(* CODESYS project RobotLibrary.library
   Company: Thorsten Brach
   Description: SRCI Robot Library
   Version: 0.0.0.36
   Placeholder: RobotLibrary
   Author: Thorsten Brach
   Title: RobotLibrary

Project tree, tasks and I/O mapping:
  libraries: RobotLibrarySysDep, 0.0.0.1 (Thorsten Brach); Tc2_Standard, 3.4.5.0 (Beckhoff Automation GmbH)
  Library/
    Constants/
      global variables RobotLibraryConstants
      global variables RobotLibraryDefines
      global variables RobotLibraryEvents
    Enumerations/
      ArmConfig/
        data type ArmConfigElbow
        data type ArmConfigShoulder
        data type ArmConfigWrist
      Events/
        data type RobotLibraryErrorIdEnum
        data type RobotLibraryInfoIdEnum
        data type RobotLibraryWarningIdEnum
      Flag/
        data type SequenceFlag
      Level/
        data type LogLevel
        data type LogLevelEnum
        data type MessageLevel
        data type PriorityLevel
      Miscellaneous/
        data type CircPlane
        data type ControlHalfByte
        data type ErrorReaction
        data type LoadMeasurementSteps
        data type PathChoice
        data type ReferenceElement
        data type Severity
        data type SyncDirection
        data type SyncReaction
        data type TriggerCondition
      Mode/
        data type AbortingMode
        data type BlendingMode
        data type CircMode
        data type CollisionReactionMode
        data type ConnectionMode
        data type DefinitionMode
        data type DetectionMode
        data type ErrorTriggerMode
        data type ExecutionMode
        data type FrameCalculationMode
        data type FunctionMode
        data type InterpolationMode
        data type JogMode
        data type LimitMode
        data type LoadMeasurementMode
        data type LogonMode
        data type MeasuringIoMode
        data type MeasuringUnitMode
        data type OperationMode
        data type OrientationMode
        data type OriMode
        data type ProcessingMode
        data type ResistanceForceMode
        data type ReturnMode
        data type SensorConnectionMode
        data type SingularityAvoidanceMode
        data type SplineMode
        data type StepMode
        data type StopMode
        data type SyncInMode
        data type SyncMode
        data type ThresholdMode
        data type ToolCalculationMode
        data type TrajectoryMode
        data type TransformMode
        data type TriggerModeIo
        data type TriggerModeLimit
        data type TriggerModeMeasurement
        data type TriggerReactionMode
        data type TurnMode
        data type WorkAreaReactionMode
      State/
        data type ActiveCommandRegisterState
        data type BufferStateCmd
        data type BufferStateRsp
        data type CmdMessageState
        data type FsmState
        data type InitializationState
        data type RaPowerState
        data type RaSequenceState
        data type RiState
        data type TelegramState
      Type/
        data type AreaType
        data type AxesGroupParameterCmdEntries
        data type CmdType
        data type ConveyorType
        data type MessageType
        data type ReferenceType
        data type UnitType
    Functions/
      Common/
        function CheckTimeout [ST]
        function SetTimeout [ST]
      Convert/
        DT/
          function DATE_TO_IEC_DATE [ST]
          function IEC_DATE_TO_DATE [ST]
          function IEC_TIME_TO_TIME [ST]
          function IEC_TIMESTAMP_TO_DT [ST]
          function TIME_TO_IEC_TIME [ST]
        Misc/
          function ArmConfigParameterToBytes [ST]
          function BytesToRCSupportedFunctions [ST]
          function ByteToFragmentAction [ST]
          function ByteToVersion [ST]
          function CombineBytesToUint [ST]
          function CombineHalfBytes [ST]
          function CombineHalfSints [ST]
          function DwordToRaStatusWord [ST]
          function FragmentActionToByte [ST]
          function PERCENT_INT_TO_REAL [ST]
          function PlcOptionalCyclicToUint [ST]
          function REAL_TO_PERCENT_INT [ST]
          function REAL_TO_PERCENT_UINT [ST]
          function RobOptionalCyclicToUint [ST]
          function VersionToByte [ST]
          function WordToArmConfigElbow [ST]
          function WordToArmConfigShoulder [ST]
          function WordToArmConfigWrist [ST]
        TO_STRING/
          function AREA_TYPE_TO_STRING [ST]
          function ARM_CONFIG_ELBOW_TO_STRING [ST]
          function ARM_CONFIG_SHOULDER_TO_STRING [ST]
          function ARM_CONFIG_TO_STRING [ST]
          function ARM_CONFIG_WRIST_TO_STRING [ST]
          function BLENDING_MODE_TO_STRING [ST]
          function BYTE_TO_STRING_BIN [ST]
          function CIRC_MODE_TO_STRING [ST]
          function CIRC_PLANE_TO_STRING [ST]
          function CMD_MESSAGE_STATE_TO_STRING [ST]
          function CMD_TYPE_TO_STRING [ST]
          function COLLISION_REACTION_MODE_TO_STRING [ST]
          function CONNECTION_MODE_TO_STRING [ST]
          function CONVEYOR_TYPE_TO_STRING [ST]
          function DATA_ENABLE_SYNC_TO_STRING [ST]
          function DATA_IN_SYNC_TO_STRING [ST]
          function DEFINITION_MODE_TO_STRING [ST]
          function DETECTION_MODE_TO_STRING [ST]
          function ERROR_REACTION_TO_STRING [ST]
          function ERROR_TRIGGER_MODE_TO_STRING [ST]
          function EXECUTION_MODE_TO_STRING [ST]
          function FRAGMENT_ACTION_TO_STRING [ST]
          function FRAME_CALCULATION_MODE_TO_STRING [ST]
          function IEC_DATE_TO_STRING [ST]
          function IEC_TIME_TO_STRING [ST]
          function INTERPOLATION_MODE_TO_STRING [ST]
          function JOG_MODE_TO_STRING [ST]
          function LIMIT_MODE_TO_STRING [ST]
          function LOAD_MEASUREMENT_MODE_TO_STRING [ST]
          function LOAD_MEASUREMENT_STEPS_TO_STRING [ST]
          function LOG_LEVEL_TO_STRING [ST]
          function LOGON_MODE_TO_STRING [ST]
          function MEASUREING_UNIT_MODE_TO_STRING [ST]
          function MESSAGE_TYPE_TO_STRING [ST]
          function ORI_MODE_TO_STRING [ST]
          function REFERENCE_TYPE_TO_STRING [ST]
          function SENSOR_CONNECTION_MODE_TO_STRING [ST]
          function SEVERITY_TO_STRING [ST]
          function SINGULARITY_AVOIDANCE_MODE_TO_STRING [ST]
          function SPLINE_MODE_TO_STRING [ST]
          function STEP_MODE_TO_STRING [ST]
          function STOP_MODE_TO_STRING [ST]
          function SYNC_IN_MODE_TO_STRING [ST]
          function SYNC_REACTION_TO_STRING [ST]
          function TELEGRAM_CONTROL_TO_STRING [ST]
          function TELEGRAM_STATE_TO_STRING [ST]
          function THRESHOLD_MODE_TO_STRING [ST]
          function TOOL_CALCULATION_MODE_TO_STRING [ST]
          function TRANSFORM_MODE_TO_STRING [ST]
          function TRIGGER_CONDITION_TO_STRING [ST]
          function TRIGGER_MODE_IO_TO_STRING [ST]
          function TRIGGER_MODE_MEASUREMENT_TO_STRING [ST]
          function TRIGGER_REACTION_MODE_TO_STRING [ST]
          function TURN_MODE_TO_STRING [ST]
          function WORD_TO_STRING_BIN [ST]
          function WORD_TO_STRING_HEX [ST]
          function WORK_AREA_REACTION_MODE_TO_STRING [ST]
      String/
        function StrPadRight [ST]
        function StrReplace [ST]
      Swap/
        function GetHalfeByteHi [ST]
        function GetHalfeByteLo [ST]
        function SwapBytes [ST]
        function SwapDword [ST]
        function SwapIecDate [ST]
        function SwapIecTime [ST]
        function SwapInt [ST]
        function SwapReal [ST]
        function SwapUdint [ST]
        function SwapUint [ST]
        function SwapWord [ST]
    Interfaces/
      interface IMessageLogger: AddMessageLog, AddSystemLog
      interface IRobotLibraryCommandFB: CallBack, CommandData
    Parameter/
      global variables RobotLibraryParameter
    POUs/
      _internal/
        function block ActiveCommandRegisterFB [ST]: AddCmd, AddRsp, CreateUniqueID, FB_init, ManageRegister, NotifyParameterChanged, OnOnlineChange, RemoveCmd, UpdateExecutionOrderList
        function block AxesGroupMessageLogFB [ST]: AddMessage, AddSystemLog, DeleteMessages, DeleteSystemLogs
        function block RobotLibraryBaseEnableFB [ST]: FSM, OnCall, OnExecCancel, OnExecErrorClear, OnExecRun, OnExecStart, Reset
        function block RobotLibraryBaseExecuteFB [ST]: FSM, OnCall, OnExecCancel, OnExecErrorClear, OnExecRun, OnExecStart, Reset
        function block RobotLibraryBaseFB [ST]: CallBack, CheckFunctionSupported, CheckParameterChanged, CheckParameterValid, CreateCommandPayload, OnCall, OnOnlineChange, ParseResponsePayload, Reset
        function block RobotLibraryLogFB [ST]: CreateLogMessage, CreateLogMessagePara1, CreateLogMessagePara2, CreateLogMessagePara3, CreateLogMessagePara4, CreateLogMessagePara5, CreateLogMessagePara6, MyType
        function block RobotLibraryRecvDataFB [ST]: GetArmConfig, GetBool, GetByte, GetDataBlock, GetDataInSync, GetDword, GetFragmentAction, GetHalfeByte1, GetHalfeByte2, GetIecDate, GetIecTime, GetInt, GetReal, GetSint, GetString, GetTrackingStatus, GetTurnNumbers, GetUdint, GetUint, GetUsint, GetWord, Reset
        function block RobotLibrarySendDataFB [ST]: AddArmConfig, AddBool, AddByte, AddDataBlock, AddDataEnableSync, AddDataInSync, AddDword, AddHalfBytes, AddIecDate, AddIecTime, AddInt, AddReal, AddSint, AddString, AddTime, AddTurnNumber, AddUdint, AddUint, AddUsint, Reset
      Additional/
        MC_AbortMeasuringInput/
          Structures/
            data type AbortMeasuringInputOutCmd
            data type AbortMeasuringInputParCmd
            data type AbortMeasuringInputRecvData
            data type AbortMeasuringInputSendData
          function block MC_AbortMeasuringInputFB [ST]: CheckFunctionSupported, CheckParameterChanged, CreateCommandPayload, CreateCommandPayloadLog, FB_init, OnCall, ParseResponsePayload, ParseResponsePayloadLog, Reset
        MC_ActivateNextCommand/
          Structures/
            data type ActivateNextCommandOutCmd
            data type ActivateNextCommandParCmd
            data type ActivateNextCommandRecvData
            data type ActivateNextCommandSendData
          function block MC_ActivateNextCommandFB [ST]: CheckFunctionSupported, CheckParameterChanged, CreateCommandPayload, CreateCommandPayloadLog, FB_init, OnCall, ParseResponsePayload, ParseResponsePayloadLog, Reset
        MC_AvoidSingularity/
          Structures/
            data type AvoidSingularityOutCmd
            data type AvoidSingularityParCmd
            data type AvoidSingularityRecvData
            data type AvoidSingularitySendData
          function block MC_AvoidSingularityFB [ST]: CheckFunctionSupported, CheckParameterChanged, CreateCommandPayload, CreateCommandPayloadLog, FB_init, OnCall, ParseResponsePayload, ParseResponsePayloadLog, Reset
        MC_BrakeTest/
          Structures/
            data type BrakeTestOutCmd
            data type BrakeTestParCmd
            data type BrakeTestRecvData
            data type BrakeTestSendData
          function block MC_BrakeTestFB [ST]: CheckFunctionSupported, CheckParameterChanged, CreateCommandPayload, CreateCommandPayloadLog, FB_init, OnCall, ParseResponsePayload, ParseResponsePayloadLog, Reset
        MC_CallSubprogram/
          Structures/
            data type CallSubprogramOutCmd
            data type CallSubprogramParCmd
            data type CallSubprogramRecvData
            data type CallSubprogramSendData
          function block MC_CallSubprogramFB [ST]: CheckFunctionSupported, CheckParameterChanged, CreateCommandPayload, CreateCommandPayloadLog, FB_init, OnCall, ParseResponsePayload, ParseResponsePayloadLog, Reset
        MC_CollisionDetection/
          Structures/
            data type CollisionDetectionOutCmd
            data type CollisionDetectionParCmd
            data type CollisionDetectionRecvData
            data type CollisionDetectionSendData
          function block MC_CollisionDetectionFB [ST]: CheckFunctionSupported, CheckParameterChanged, CreateCommandPayload, CreateCommandPayloadLog, FB_init, OnCall, ParseResponsePayload, ParseResponsePayloadLog, Reset
        MC_ExchangeConfiguration/
          Structures/
            data type ExchangeConfigurationOutCmd
            data type ExchangeConfigurationParCmd
            data type ExchangeConfigurationRecvData
            data type ExchangeConfigurationSendData
          function block MC_ExchangeConfigurationFB [ST]: CheckFunctionSupported, CheckParameterChanged, CreateCommandPayload, CreateCommandPayloadLog, FB_init, OnCall, ParseResponsePayload, ParseResponsePayloadLog, Reset
        MC_FreeDrive/
          Structures/
            data type FreeDriveOutCmd
            data type FreeDriveParCmd
            data type FreeDriveRecvData
            data type FreeDriveSendData
          function block MC_FreeDriveFB [ST]: CheckFunctionSupported, CheckParameterChanged, CreateCommandPayload, CreateCommandPayloadLog, FB_init, OnCall, ParseResponsePayload, ParseResponsePayloadLog, Reset
        MC_MeasuringInput/
          Structures/
            data type MeasuringInputOutCmd
            data type MeasuringInputParCmd
            data type MeasuringInputRecvData
            data type MeasuringInputSendData
          function block MC_MeasuringInputFB [ST]: CheckFunctionSupported, CheckParameterChanged, CreateCommandPayload, CreateCommandPayloadLog, FB_init, OnCall, ParseResponsePayload, ParseResponsePayloadLog, Reset
        MC_OpenBrake/
          Structures/
            data type OpenBrakeOutCmd
            data type OpenBrakeParCmd
            data type OpenBrakeRecvData
            data type OpenBrakeSendData
          function block MC_OpenBrakeFB [ST]: CheckFunctionSupported, CheckParameterChanged, CreateCommandPayload, CreateCommandPayloadLog, FB_init, OnCall, ParseResponsePayload, ParseResponsePayloadLog, Reset
        MC_PathAccuracyMode/
          Structures/
            data type PathAccuracyModeOutCmd
            data type PathAccuracyModeParCmd
            data type PathAccuracyModeRecvData
            data type PathAccuracyModeSendData
          function block MC_PathAccuracyModeFB [ST]: CheckFunctionSupported, CheckParameterChanged, CreateCommandPayload, CreateCommandPayloadLog, FB_init, OnCall, ParseResponsePayload, ParseResponsePayloadLog, Reset
        MC_ReadCallSubprogramCyclic/
          Structures/
            data type ReadCallSubprogramCyclicOutCmd
            data type ReadCallSubprogramCyclicParCmd
          function block MC_ReadCallSubprogramCyclicFB [ST]: CheckFunctionSupported, FB_init, OnCall
        MC_ShiftPosition/
          Structures/
            data type ShiftPositionOutCmd
            data type ShiftPositionParCmd
            data type ShiftPositionRecvData
            data type ShiftPositionSendData
          function block MC_ShiftPositionFB [ST]: CheckFunctionSupported, CheckParameterChanged, CreateCommandPayload, CreateCommandPayloadLog, FB_init, OnCall, ParseResponsePayload, ParseResponsePayloadLog, Reset
        MC_SoftSwitchTcp/
          Structures/
            data type SoftSwitchTcpOutCmd
            data type SoftSwitchTcpParCmd
            data type SoftSwitchTcpRecvData
            data type SoftSwitchTcpSendData
          function block MC_SoftSwitchTcpFB [ST]: CheckFunctionSupported, CheckParameterChanged, CreateCommandPayload, CreateCommandPayloadLog, FB_init, OnCall, ParseResponsePayload, ParseResponsePayloadLog, Reset
        MC_StopSubprogram/
          Structures/
            data type StopSubprogramOutCmd
            data type StopSubprogramParCmd
            data type StopSubprogramRecvData
            data type StopSubprogramSendData
          function block MC_StopSubprogramFB [ST]: CheckFunctionSupported, CheckParameterChanged, CreateCommandPayload, CreateCommandPayloadLog, FB_init, OnCall, ParseResponsePayload, ParseResponsePayloadLog, Reset
        MC_UnitMeasurement/
          Structures/
            data type UnitMeasurementOutCmd
            data type UnitMeasurementParCmd
            data type UnitMeasurementRecvData
            data type UnitMeasurementSendData
          function block MC_UnitMeasurementFB [ST]: CheckFunctionSupported, CheckParameterChanged, CreateCommandPayload, CreateCommandPayloadLog, FB_init, OnCall, ParseResponsePayload, ParseResponsePayloadLog, Reset
        MC_WriteCallSubprogramCyclic/
          Structures/
            data type WriteCallSubprogramCyclicOutCmd
            data type WriteCallSubprogramCyclicParCmd
          function block MC_WriteCallSubprogramCyclicFB [ST]: CheckFunctionSupported, FB_init, OnCall
      AdvancedMove/
        MC_MoveApproachDirect/
          Structures/
            data type MoveApproachDirectOutCmd
            data type MoveApproachDirectParCmd
            data type MoveApproachDirectRecvData
            data type MoveApproachDirectSendData
          function block MC_MoveApproachDirectFB [ST]: CheckFunctionSupported, CheckParameterChanged, CreateCommandPayload, CreateCommandPayloadLog, FB_init, OnCall, ParseResponsePayload, ParseResponsePayloadLog, Reset
        MC_MoveApproachLinear/
          Structures/
            data type MoveApproachLinearOutCmd
            data type MoveApproachLinearParCmd
            data type MoveApproachLinearRecvData
            data type MoveApproachLinearSendData
          function block MC_MoveApproachLinearFB [ST]: CheckFunctionSupported, CheckParameterChanged, CreateCommandPayload, CreateCommandPayloadLog, FB_init, OnCall, ParseResponsePayload, ParseResponsePayloadLog, Reset
        MC_MoveAxesRelative/
          Structures/
            data type MoveAxesRelativeOutCmd
            data type MoveAxesRelativeParCmd
            data type MoveAxesRelativeRecvData
            data type MoveAxesRelativeSendData
          function block MC_MoveAxesRelativeFB [ST]: CheckFunctionSupported, CheckParameterChanged, CreateCommandPayload, CreateCommandPayloadLog, FB_init, OnCall, ParseResponsePayload, ParseResponsePayloadLog, Reset
        MC_MoveCircularAbsolute/
          Structures/
            data type MoveCircularAbsoluteOutCmd
            data type MoveCircularAbsoluteParCmd
            data type MoveCircularAbsoluteRecvData
            data type MoveCircularAbsoluteSendData
          function block MC_MoveCircularAbsoluteFB [ST]: CheckFunctionSupported, CheckParameterChanged, CreateCommandPayload, CreateCommandPayloadLog, FB_init, OnCall, ParseResponsePayload, ParseResponsePayloadLog, Reset
        MC_MoveCircularCamFB/
          Structures/
            data type MoveCircularCamOutCmd
            data type MoveCircularCamParCmd
            data type MoveCircularCamRecvData
            data type MoveCircularCamSendData
          function block MC_MoveCircularCamFB [ST]: CheckFunctionSupported, CheckParameterChanged, CreateCommandPayload, CreateCommandPayloadLog, FB_init, OnCall, ParseResponsePayload, ParseResponsePayloadLog, Reset
        MC_MoveCircularRelative/
          Structures/
            data type MoveCircularRelativeOutCmd
            data type MoveCircularRelativeParCmd
            data type MoveCircularRelativeRecvData
            data type MoveCircularRelativeSendData
          function block MC_MoveCircularRelativeFB [ST]: CheckFunctionSupported, CheckParameterChanged, CreateCommandPayload, CreateCommandPayloadLog, FB_init, OnCall, ParseResponsePayload, ParseResponsePayloadLog, Reset
        MC_MoveDepartDirect/
          Structures/
            data type MoveDepartDirectOutCmd
            data type MoveDepartDirectParCmd
            data type MoveDepartDirectRecvData
            data type MoveDepartDirectSendData
          function block MC_MoveDepartDirectFB [ST]: CheckFunctionSupported, CheckParameterChanged, CreateCommandPayload, CreateCommandPayloadLog, FB_init, OnCall, ParseResponsePayload, ParseResponsePayloadLog, Reset
        MC_MoveDepartLinear/
          Structures/
            data type MoveDepartLinearOutCmd
            data type MoveDepartLinearParCmd
            data type MoveDepartLinearRecvData
            data type MoveDepartLinearSendData
          function block MC_MoveDepartLinearFB [ST]: CheckFunctionSupported, CheckParameterChanged, CreateCommandPayload, CreateCommandPayloadLog, FB_init, OnCall, ParseResponsePayload, ParseResponsePayloadLog, Reset
        MC_MoveDirectOffset/
          Structures/
            data type MoveDirectOffsetOutCmd
            data type MoveDirectOffsetParCmd
            data type MoveDirectOffsetRecvData
            data type MoveDirectOffsetSendData
          function block MC_MoveDirectOffsetFB [ST]: CheckFunctionSupported, CheckParameterChanged, CreateCommandPayload, CreateCommandPayloadLog, FB_init, OnCall, ParseResponsePayload, ParseResponsePayloadLog, Reset
        MC_MoveDirectRelative/
          Structures/
            data type MoveDirectRelativeOutCmd
            data type MoveDirectRelativeParCmd
            data type MoveDirectRelativeRecvData
            data type MoveDirectRelativeSendData
          function block MC_MoveDirectRelativeFB [ST]: CheckFunctionSupported, CheckParameterChanged, CreateCommandPayload, CreateCommandPayloadLog, FB_init, OnCall, ParseResponsePayload, ParseResponsePayloadLog, Reset
        MC_MoveLinearAbsoluteJ/
          Structures/
            data type MoveLinearAbsoluteJOutCmd
            data type MoveLinearAbsoluteJParCmd
            data type MoveLinearAbsoluteJRecvData
            data type MoveLinearAbsoluteJSendData
          function block MC_MoveLinearAbsoluteJFB [ST]: CheckFunctionSupported, CheckParameterChanged, CreateCommandPayload, CreateCommandPayloadLog, FB_init, OnCall, ParseResponsePayload, ParseResponsePayloadLog, Reset
        MC_MoveLinearCam/
          Structures/
            data type MoveLinearCamOutCmd
            data type MoveLinearCamParCmd
            data type MoveLinearCamRecvData
            data type MoveLinearCamSendData
          function block MC_MoveLinearCamFB [ST]: CheckFunctionSupported, CheckParameterChanged, CreateCommandPayload, CreateCommandPayloadLog, FB_init, OnCall, ParseResponsePayload, ParseResponsePayloadLog, Reset
        MC_MoveLinearOffset/
          Structures/
            data type MoveLinearOffsetOutCmd
            data type MoveLinearOffsetParCmd
            data type MoveLinearOffsetRecvData
            data type MoveLinearOffsetSendData
          function block MC_MoveLinearOffsetFB [ST]: CheckFunctionSupported, CheckParameterChanged, CreateCommandPayload, CreateCommandPayloadLog, FB_init, OnCall, ParseResponsePayload, ParseResponsePayloadLog, Reset
        MC_MoveLinearRelative/
          Structures/
            data type MoveLinearRelativeOutCmd
            data type MoveLinearRelativeParCmd
            data type MoveLinearRelativeRecvData
            data type MoveLinearRelativeSendData
          function block MC_MoveLinearRelativeFB [ST]: CheckFunctionSupported, CheckParameterChanged, CreateCommandPayload, CreateCommandPayloadLog, FB_init, OnCall, ParseResponsePayload, ParseResponsePayloadLog, Reset
        MC_MovePickPlaceDirect/
          Structures/
            data type MovePickPlaceDirectOutCmd
            data type MovePickPlaceDirectParCmd
            data type MovePickPlaceDirectRecvData
            data type MovePickPlaceDirectSendData
          function block MC_MovePickPlaceDirectFB [ST]: CheckFunctionSupported, CheckParameterChanged, CreateCommandPayload, CreateCommandPayloadLog, FB_init, OnCall, ParseResponsePayload, ParseResponsePayloadLog, Reset
        MC_MovePickPlaceLinear/
          Structures/
            data type MovePickPlaceLinearOutCmd
            data type MovePickPlaceLinearParCmd
            data type MovePickPlaceLinearRecvData
            data type MovePickPlaceLinearSendData
          function block MC_MovePickPlaceLinearFB [ST]: CheckFunctionSupported, CheckParameterChanged, CreateCommandPayload, CreateCommandPayloadLog, FB_init, OnCall, ParseResponsePayload, ParseResponsePayloadLog, Reset
      BasicMove/
        MC_ChangeSpeedOverride/
          Structures/
            data type ChangeSpeedOverrideOutCmd
            data type ChangeSpeedOverrideParCmd
            data type ChangeSpeedOverrideRecvData
            data type ChangeSpeedOverrideSendData
          function block MC_ChangeSpeedOverrideFB [ST]: CheckFunctionSupported, CheckParameterChanged, CreateCommandPayload, CreateCommandPayloadLog, FB_init, OnCall, ParseResponsePayload, ParseResponsePayloadLog, Reset
        MC_GroupContinue/
          Structures/
            data type GroupContinueOutCmd
            data type GroupContinueParCmd
            data type GroupContinueRecvData
            data type GroupContinueSendData
          function block MC_GroupContinueFB [ST]: CheckFunctionSupported, CheckParameterChanged, CreateCommandPayload, CreateCommandPayloadLog, FB_init, OnCall, ParseResponsePayload, ParseResponsePayloadLog, Reset
        MC_GroupInterrupt/
          Structures/
            data type GroupInterruptOutCmd
            data type GroupInterruptParCmd
            data type GroupInterruptRecvData
            data type GroupInterruptSendData
          function block MC_GroupInterruptFB [ST]: CheckFunctionSupported, CheckParameterChanged, CreateCommandPayload, CreateCommandPayloadLog, FB_init, OnCall, ParseResponsePayload, ParseResponsePayloadLog, Reset
        MC_GroupJog/
          Structures/
            data type GroupJogOutCmd
            data type GroupJogParCmd
            data type GroupJogRecvData
            data type GroupJogSendData
          function block MC_GroupJogFB [ST]: CheckFunctionSupported, CheckParameterChanged, CreateCommandPayload, CreateCommandPayloadLog, FB_init, OnCall, ParseResponsePayload, ParseResponsePayloadLog, Reset
        MC_GroupStop/
          Structures/
            data type GroupStopOutCmd
            data type GroupStopParCmd
            data type GroupStopRecvData
            data type GroupStopSendData
          function block MC_GroupStopFB [ST]: CheckFunctionSupported, CheckParameterChanged, CreateCommandPayload, CreateCommandPayloadLog, FB_init, OnCall, ParseResponsePayload, ParseResponsePayloadLog, Reset
        MC_MoveAxesAbsolute/
          Structures/
            data type MoveAxesAbsoluteOutCmd
            data type MoveAxesAbsoluteParCmd
            data type MoveAxesAbsoluteRecvData
            data type MoveAxesAbsoluteSendData
          function block MC_MoveAxesAbsoluteFB [ST]: CheckFunctionSupported, CheckParameterChanged, CreateCommandPayload, CreateCommandPayloadLog, FB_init, OnCall, ParseResponsePayload, ParseResponsePayloadLog, Reset
        MC_MoveDirectAbsolute/
          Structures/
            data type MoveDirectAbsoluteOutCmd
            data type MoveDirectAbsoluteParCmd
            data type MoveDirectAbsoluteRecvData
            data type MoveDirectAbsoluteSendData
          function block MC_MoveDirectAbsoluteFB [ST]: CheckFunctionSupported, CheckParameterChanged, CreateCommandPayload, CreateCommandPayloadLog, FB_init, OnCall, ParseResponsePayload, ParseResponsePayloadLog, Reset
        MC_MoveLinearAbsolute/
          Structures/
            data type MoveLinearAbsoluteOutCmd
            data type MoveLinearAbsoluteParCmd
            data type MoveLinearAbsoluteRecvData
            data type MoveLinearAbsoluteSendData
          function block MC_MoveLinearAbsoluteFB [ST]: CheckFunctionSupported, CheckParameterChanged, CreateCommandPayload, CreateCommandPayloadLog, FB_init, OnCall, ParseResponsePayload, ParseResponsePayloadLog, Reset
        MC_ReturnToPrimary/
          Structures/
            data type ReturnToPrimaryOutCmd
            data type ReturnToPrimaryParCmd
            data type ReturnToPrimaryRecvData
            data type ReturnToPrimarySendData
          function block MC_ReturnToPrimaryFB [ST]: CheckFunctionSupported, CheckParameterChanged, CreateCommandPayload, CreateCommandPayloadLog, FB_init, OnCall, ParseResponsePayload, ParseResponsePayloadLog, Reset
      Calculation/
        MC_CalculateCartesianPosition/
          Structures/
            data type CalculateCartesianPositionOutCmd
            data type CalculateCartesianPositionParCmd
            data type CalculateCartesianPositionRecvData
            data type CalculateCartesianPositionSendData
          function block MC_CalculateCartesianPositionFB [ST]: CheckFunctionSupported, CheckParameterChanged, CreateCommandPayload, CreateCommandPayloadLog, FB_init, OnCall, ParseResponsePayload, ParseResponsePayloadLog, Reset
        MC_CalculateForwardKinematic/
          Structures/
            data type CalculateForwardKinematicOutCmd
            data type CalculateForwardKinematicParCmd
            data type CalculateForwardKinematicRecvData
            data type CalculateForwardKinematicSendData
          function block MC_CalculateForwardKinematicFB [ST]: CheckFunctionSupported, CheckParameterChanged, CreateCommandPayload, CreateCommandPayloadLog, FB_init, OnCall, ParseResponsePayload, ParseResponsePayloadLog, Reset
        MC_CalculateFrame/
          Structures/
            data type CalculateFrameOutCmd
            data type CalculateFrameParCmd
            data type CalculateFrameRecvData
            data type CalculateFrameSendData
          function block MC_CalculateFrameFB [ST]: CheckFunctionSupported, CheckParameterChanged, CreateCommandPayload, CreateCommandPayloadLog, FB_init, OnCall, ParseResponsePayload, ParseResponsePayloadLog, Reset
        MC_CalculateInverseKinematic/
          Structures/
            data type CalculateInverseKinematicOutCmd
            data type CalculateInverseKinematicParCmd
            data type CalculateInverseKinematicRecvData
            data type CalculateInverseKinematicSendData
          function block MC_CalculateInverseKinematicFB [ST]: CheckFunctionSupported, CheckParameterChanged, CreateCommandPayload, CreateCommandPayloadLog, FB_init, OnCall, ParseResponsePayload, ParseResponsePayloadLog, Reset
        MC_CalculateTool/
          Structures/
            data type CalculateToolOutCmd
            data type CalculateToolParCmd
            data type CalculateToolRecvData
            data type CalculateToolSendData
          function block MC_CalculateToolFB [ST]: CheckFunctionSupported, CheckParameterChanged, CreateCommandPayload, CreateCommandPayloadLog, FB_init, OnCall, ParseResponsePayload, ParseResponsePayloadLog, Reset
        MC_LoadMeasurementAutomatic/
          Structures/
            data type LoadMeasurementAutomaticOutCmd
            data type LoadMeasurementAutomaticParCmd
            data type LoadMeasurementAutomaticRecvData
            data type LoadMeasurementAutomaticSendData
          function block MC_LoadMeasurementAutomaticFB [ST]: CheckFunctionSupported, CheckParameterChanged, CreateCommandPayload, CreateCommandPayloadLog, FB_init, OnCall, ParseResponsePayload, ParseResponsePayloadLog, Reset
        MC_LoadMeasurementSequential/
          Structures/
            data type LoadMeasurementSequentialOutCmd
            data type LoadMeasurementSequentialParCmd
            data type LoadMeasurementSequentialRecvData
            data type LoadMeasurementSequentialSendData
          function block MC_LoadMeasurementSequentialFB [ST]: CheckFunctionSupported, CheckParameterChanged, CreateCommandPayload, CreateCommandPayloadLog, FB_init, OnCall, ParseResponsePayload, ParseResponsePayloadLog, Reset
      ConveyorTracking/
        MC_ActivateConveyorTracking/
          Structures/
            data type ActivateConveyorTrackingOutCmd
            data type ActivateConveyorTrackingParCmd
            data type ActivateConveyorTrackingRecvData
            data type ActivateConveyorTrackingSendData
          function block MC_ActivateConveyorTrackingFB [ST]: CheckFunctionSupported, CheckParameterChanged, CreateCommandPayload, CreateCommandPayloadLog, FB_init, OnCall, ParseResponsePayload, ParseResponsePayloadLog, Reset
        MC_ConfigureConveyor/
          Structures/
            data type ConfigureConveyorOutCmd
            data type ConfigureConveyorParCmd
            data type ConfigureConveyorRecvData
            data type ConfigureConveyorSendData
          function block MC_ConfigureConveyorFB [ST]: CheckFunctionSupported, CheckParameterChanged, CreateCommandPayload, CreateCommandPayloadLog, FB_init, OnCall, ParseResponsePayload, ParseResponsePayloadLog, Reset
        MC_RedefineTrackingPos/
          Structures/
            data type RedefineTrackingPosOutCmd
            data type RedefineTrackingPosParCmd
            data type RedefineTrackingPosRecvData
            data type RedefineTrackingPosSendData
          function block MC_RedefineTrackingPosFB [ST]: CheckFunctionSupported, CheckParameterChanged, CreateCommandPayload, CreateCommandPayloadLog, FB_init, OnCall, ParseResponsePayload, ParseResponsePayloadLog, Reset
        MC_SyncToConveyor/
          Structures/
            data type SyncToConveyorOutCmd
            data type SyncToConveyorParCmd
            data type SyncToConveyorRecvData
            data type SyncToConveyorSendData
          function block MC_SyncToConveyorFB [ST]: CheckFunctionSupported, CheckParameterChanged, CreateCommandPayload, CreateCommandPayloadLog, FB_init, OnCall, ParseResponsePayload, ParseResponsePayloadLog, Reset
      ForceControl/
        MC_ForceControl/
          Structures/
            data type ForceControlOutCmd
            data type ForceControlParCmd
            data type ForceControlRecvData
            data type ForceControlSendData
          function block MC_ForceControlFB [ST]: CheckFunctionSupported, CheckParameterChanged, CreateCommandPayload, CreateCommandPayloadLog, FB_init, OnCall, ParseResponsePayload, ParseResponsePayloadLog, Reset
        MC_ForceLimit/
          Structures/
            data type ForceLimitOutCmd
            data type ForceLimitParCmd
            data type ForceLimitRecvData
            data type ForceLimitSendData
          function block MC_ForceLimitFB [ST]: CheckFunctionSupported, CheckParameterChanged, CreateCommandPayload, CreateCommandPayloadLog, FB_init, OnCall, ParseResponsePayload, ParseResponsePayloadLog, Reset
        MC_ReadActualForce/
          Structures/
            data type ReadActualForceOutCmd
            data type ReadActualForceParCmd
            data type ReadActualForceRecvData
            data type ReadActualForceSendData
          function block MC_ReadActualForceFB [ST]: CheckFunctionSupported, CheckParameterChanged, CreateCommandPayload, CreateCommandPayloadLog, FB_init, OnCall, ParseResponsePayload, ParseResponsePayloadLog, Reset
      General/
        MC_CreateServerLog_ToDo/
          function block MC_CreateServerLog_ToDo [ST]: FB_init
        MC_EnableRobot/
          Structures/
            data type EnableRobotOutCmd
            data type EnableRobotParCmd
            data type EnableRobotRecvData
            data type EnableRobotSendData
          function block MC_EnableRobotFB [ST]: CheckFunctionSupported, CheckParameterChanged, CreateCommandPayload, CreateCommandPayloadLog, FB_init, OnCall, ParseResponsePayload, ParseResponsePayloadLog, Reset
        MC_GroupReset/
          Structures/
            data type GroupResetOutCmd
            data type GroupResetParCmd
            data type GroupResetRecvData
            data type GroupResetSendData
          function block MC_GroupResetFB [ST]: CheckFunctionSupported, CheckParameterChanged, CreateCommandPayload, CreateCommandPayloadLog, FB_init, OnCall, ParseResponsePayload, ParseResponsePayloadLog, Reset
        MC_ReadServerLog_ToDo/
          function block MC_ReadServerLog [ST]: FB_init
        MC_RestartController/
          Structures/
            data type RestartControllerOutCmd
            data type RestartControllerParCmd
            data type RestartControllerRecvData
            data type RestartControllerSendData
          function block MC_RestartControllerFB [ST]: CheckFunctionSupported, CheckParameterChanged, CreateCommandPayload, CreateCommandPayloadLog, FB_init, OnCall, ParseResponsePayload, ParseResponsePayloadLog, Reset
        MC_RobotTask/
          Structures/
            ParCfg/
              Com/
                data type RobotTaskParCfgCom
              Plc/
                data type RobotTaskParCfgPlc
                data type RobotTaskParCfgPlcParameter
              Rob/
                data type RobotTaskParCfgRob
                data type RobotTaskParCfgRobParameter
              data type RobotTaskParCfg
          function block MC_RobotTaskFB [ST]: AxesGroupFromTelegram, AxesGroupFromTelegramCyclic, AxesGroupFromTelegramCyclicOptional, AxesGroupToTelegram, AxesGroupToTelegramCyclic, AxesGroupToTelegramCyclicOptional, AxesGroupToTelegramFooter, AxesGroupToTelegramHeader, AxesGroupToTelegramLogging, AxesGroupToTelegramSequence, CalcTelegramLengthPlcToRob, CreateSendPayload, CreateSendPayloadCyclic, CreateSendPayloadCyclicOptional, CreateSendPayloadFooter, CreateSendPayloadHeader, CreateSendPayloadLogging, CreateSendPayloadSequence, FB_init, HandleAliveBit, HandleAxesGroupAcyclic, HandleAxesGroupCyclic, HandleAxesGroupCyclicOptional, HandleAxesGroupInternalData, HandleAxesGroupMessageLog, HandleAxesGroupParameter, HandleAxesGroupState, HandleInvalidFrames, HandleLifeSign, HandleSeqAck, HandleTelegramStateCtrl, OnCall, OnErrorClear, OnExecRun, ParseRecvPayload, ParseRecvPayloadCyclic, ParseRecvPayloadCyclicOptional, ParseRecvPayloadFooter, ParseRecvPayloadHeader, ParseRecvPayloadLogging, ParseRecvPayloadSequence
        MC_SetOperationMode/
          Structures/
            data type SetOperationModeOutCmd
            data type SetOperationModeParCmd
            data type SetOperationModeRecvData
            data type SetOperationModeSendData
          function block MC_SetOperationModeFB [ST]: CheckFunctionSupported, CheckParameterChanged, CreateCommandPayload, CreateCommandPayloadLog, FB_init, OnCall, ParseResponsePayload, ParseResponsePayloadLog, Reset
        MC_SetSequence/
          Structures/
            data type SetSequenceOutCmd
            data type SetSequenceParCmd
            data type SetSequenceRecvData
            data type SetSequenceSendData
          function block MC_SetSequenceFB [ST]: CheckFunctionSupported, CheckParameterChanged, CreateCommandPayload, CreateCommandPayloadLog, FB_init, OnCall, ParseResponsePayload, ParseResponsePayloadLog, Reset
        MC_SwitchLanguage/
          Structures/
            data type SwitchLanguageOutCmd
            data type SwitchLanguageParCmd
            data type SwitchLanguageRecvData
            data type SwitchLanguageSendData
          function block MC_SwitchLanguageFB [ST]: CheckFunctionSupported, CheckParameterChanged, CreateCommandPayload, CreateCommandPayloadLog, FB_init, OnCall, ParseResponsePayload, ParseResponsePayloadLog, Reset
        MC_UserLogin/
          Structures/
            data type UserLoginOutCmd
            data type UserLoginParCmd
            data type UserLoginRecvData
            data type UserLoginSendData
          function block MC_UserLoginFB [ST]: CheckFunctionSupported, CheckParameterChanged, CreateCommandPayload, CreateCommandPayloadLog, FB_init, OnCall, ParseResponsePayload, ParseResponsePayloadLog, Reset
      Read/
        MC_ReadActualPosition/
          Structures/
            data type ReadActualPositionOutCmd
            data type ReadActualPositionParCmd
            data type ReadActualPositionRecvData
            data type ReadActualPositionSendData
          function block MC_ReadActualPositionFB [ST]: CheckFunctionSupported, CheckParameterChanged, CreateCommandPayload, CreateCommandPayloadLog, FB_init, OnCall, ParseResponsePayload, ParseResponsePayloadLog, Reset
        MC_ReadActualPositionCyclic/
          Structures/
            data type ReadActualPositionCyclicOutCmd
            data type ReadActualPositionCyclicParCmd
          function block MC_ReadActualPositionCyclicFB [ST]: CheckFunctionSupported, CheckParameterChanged, CheckParameterValid, CreateCommandParameterLog, FB_init, OnCall, Reset
        MC_ReadActualTCPVelocity/
          Structures/
            data type ReadActualTCPVelocityOutCmd
            data type ReadActualTCPVelocityParCmd
            data type ReadActualTCPVelocityRecvData
            data type ReadActualTCPVelocitySendData
          function block MC_ReadActualTCPVelocityFB [ST]: CheckFunctionSupported, CheckParameterChanged, CreateCommandPayload, CreateCommandPayloadLog, FB_init, OnCall, ParseResponsePayload, ParseResponsePayloadLog, Reset
        MC_ReadAnalogInput/
          Structures/
            data type ReadAnalogInputOutCmd
            data type ReadAnalogInputParCmd
            data type ReadAnalogInputRecvData
            data type ReadAnalogInputSendData
          function block MC_ReadAnalogInputFB [ST]: CheckFunctionSupported, CheckParameterChanged, CreateCommandPayload, CreateCommandPayloadLog, FB_init, OnCall, ParseResponsePayload, ParseResponsePayloadLog, Reset
        MC_ReadDHParameter/
          Structures/
            data type ReadDHParameterOutCmd
            data type ReadDHParameterParCmd
            data type ReadDHParameterRecvData
            data type ReadDHParameterSendData
          function block MC_ReadDHParameterFB [ST]: CheckFunctionSupported, CheckParameterChanged, CreateCommandPayload, CreateCommandPayloadLog, FB_init, OnCall, ParseResponsePayload, ParseResponsePayloadLog, Reset
        MC_ReadDigitalInputs/
          Structures/
            data type ReadDigitalInputsOutCmd
            data type ReadDigitalInputsParCmd
            data type ReadDigitalInputsRecvData
            data type ReadDigitalInputsSendData
          function block MC_ReadDigitalInputsFB [ST]: CheckFunctionSupported, CheckParameterChanged, CreateCommandPayload, CreateCommandPayloadLog, FB_init, OnCall, ParseResponsePayload, ParseResponsePayloadLog, Reset
        MC_ReadDigitalOutputs/
          Structures/
            data type ReadDigitalOutputsOutCmd
            data type ReadDigitalOutputsParCmd
            data type ReadDigitalOutputsRecvData
            data type ReadDigitalOutputsSendData
          function block MC_ReadDigitalOutputsFB [ST]: CheckFunctionSupported, CheckParameterChanged, CreateCommandPayload, CreateCommandPayloadLog, FB_init, OnCall, ParseResponsePayload, ParseResponsePayloadLog, Reset
        MC_ReadFrameData/
          Structures/
            data type ReadFrameDataOutCmd
            data type ReadFrameDataParCmd
            data type ReadFrameDataRecvData
            data type ReadFrameDataSendData
          function block MC_ReadFrameDataFB [ST]: CheckFunctionSupported, CheckParameterChanged, CreateCommandPayload, CreateCommandPayloadLog, FB_init, OnCall, ParseResponsePayload, ParseResponsePayloadLog, Reset
        MC_ReadIntegers/
          Structures/
            data type ReadIntegersOutCmd
            data type ReadIntegersParCmd
            data type ReadIntegersRecvData
            data type ReadIntegersSendData
          function block MC_ReadIntegersFB [ST]: CheckFunctionSupported, CheckParameterChanged, CreateCommandPayload, CreateCommandPayloadLog, FB_init, OnCall, ParseResponsePayload, ParseResponsePayloadLog, Reset
        MC_ReadLoadData/
          Structures/
            data type ReadLoadDataOutCmd
            data type ReadLoadDataParCmd
            data type ReadLoadDataRecvData
            data type ReadLoadDataSendData
          function block MC_ReadLoadDataFB [ST]: CheckFunctionSupported, CheckParameterChanged, CreateCommandPayload, CreateCommandPayloadLog, FB_init, OnCall, ParseResponsePayload, ParseResponsePayloadLog, Reset
        MC_ReadMessages/
          Structures/
            data type ReadMessagesOutCmd
            data type ReadMessagesParCmd
            data type ReadMessagesRecvData
            data type ReadMessagesSendData
          function block MC_ReadMessagesFB [ST]: CheckFunctionSupported, CheckParameterChanged, CreateCommandPayload, CreateCommandPayloadLog, FB_init, OnCall, ParseResponsePayload, ParseResponsePayloadLog, Reset
        MC_ReadReals/
          Structures/
            data type ReadRealsOutCmd
            data type ReadRealsParCmd
            data type ReadRealsRecvData
            data type ReadRealsSendData
          function block MC_ReadRealsFB [ST]: CheckFunctionSupported, CheckParameterChanged, CreateCommandPayload, CreateCommandPayloadLog, FB_init, OnCall, ParseResponsePayload, ParseResponsePayloadLog, Reset
        MC_ReadRobotData/
          Structures/
            data type ReadRobotDataOutCmd
            data type ReadRobotDataParCmd
            data type ReadRobotDataRecvData
            data type ReadRobotDataSendData
          function block MC_ReadRobotDataFB [ST]: CheckFunctionSupported, CheckParameterChanged, CreateCommandPayload, CreateCommandPayloadLog, FB_init, OnCall, ParseResponsePayload, ParseResponsePayloadLog, Reset
        MC_ReadRobotDefaultDynamics/
          Structures/
            data type ReadRobotDefaultDynamicsOutCmd
            data type ReadRobotDefaultDynamicsParCmd
            data type ReadRobotDefaultDynamicsRecvData
            data type ReadRobotDefaultDynamicsSendData
          function block MC_ReadRobotDefaultDynamicsFB [ST]: CheckFunctionSupported, CheckParameterChanged, CreateCommandPayload, CreateCommandPayloadLog, FB_init, OnCall, ParseResponsePayload, ParseResponsePayloadLog, Reset
        MC_ReadRobotReferenceDynamics/
          Structures/
            data type ReadRobotReferenceDynamicsOutCmd
            data type ReadRobotReferenceDynamicsParCmd
            data type ReadRobotReferenceDynamicsRecvData
            data type ReadRobotReferenceDynamicsSendData
          function block MC_ReadRobotReferenceDynamicsFB [ST]: CheckFunctionSupported, CheckParameterChanged, CreateCommandPayload, CreateCommandPayloadLog, FB_init, OnCall, ParseResponsePayload, ParseResponsePayloadLog, Reset
        MC_ReadRobotSWLimits/
          Structures/
            data type ReadRobotSWLimitsOutCmd
            data type ReadRobotSWLimitsParCmd
            data type ReadRobotSWLimitsRecvData
            data type ReadRobotSWLimitsSendData
          function block MC_ReadRobotSWLimitsFB [ST]: CheckFunctionSupported, CheckParameterChanged, CreateCommandPayload, CreateCommandPayloadLog, FB_init, OnCall, ParseResponsePayload, ParseResponsePayloadLog, Reset
        MC_ReadSystemVariable/
          Structures/
            data type ReadSystemVariableOutCmd
            data type ReadSystemVariableParCmd
            data type ReadSystemVariableRecvData
            data type ReadSystemVariableSendData
          function block MC_ReadSystemVariableFB [ST]: CheckFunctionSupported, CheckParameterChanged, CreateCommandPayload, CreateCommandPayloadLog, FB_init, OnCall, ParseResponsePayload, ParseResponsePayloadLog, Reset
        MC_ReadToolData/
          Structures/
            data type ReadToolDataOutCmd
            data type ReadToolDataParCmd
            data type ReadToolDataRecvData
            data type ReadToolDataSendData
          function block MC_ReadToolDataFB [ST]: CheckFunctionSupported, CheckParameterChanged, CreateCommandPayload, CreateCommandPayloadLog, FB_init, OnCall, ParseResponsePayload, ParseResponsePayloadLog, Reset
      SearchHardstop/
        MC_SearchHardStop/
          Structures/
            data type SearchHardStopOutCmd
            data type SearchHardStopParCmd
            data type SearchHardStopRecvData
            data type SearchHardStopSendData
          function block MC_SearchHardStopFB [ST]: CheckFunctionSupported, CheckParameterChanged, CreateCommandPayload, CreateCommandPayloadLog, FB_init, OnCall, ParseResponsePayload, ParseResponsePayloadLog, Reset
        MC_SearchHardStopJ/
          Structures/
            data type SearchHardStopJOutCmd
            data type SearchHardStopJParCmd
            data type SearchHardStopJRecvData
            data type SearchHardStopJSendData
          function block MC_SearchHardStopJFB [ST]: CheckFunctionSupported, CheckParameterChanged, CreateCommandPayload, CreateCommandPayloadLog, FB_init, OnCall, ParseResponsePayload, ParseResponsePayloadLog, Reset
      Spline/
        MC_CreateSpline/
          Structures/
            data type CreateSplineOutCmd
            data type CreateSplineParCmd
            data type CreateSplineRecvData
            data type CreateSplineSendData
          function block MC_CreateSplineFB [ST]: CheckFunctionSupported, CheckParameterChanged, CreateCommandPayload, CreateCommandPayloadLog, FB_init, OnCall, ParseResponsePayload, ParseResponsePayloadLog, Reset
        MC_DeleteSpline/
          Structures/
            data type DeleteSplineOutCmd
            data type DeleteSplineParCmd
            data type DeleteSplineRecvData
            data type DeleteSplineSendData
          function block MC_DeleteSplineFB [ST]: CheckFunctionSupported, CheckParameterChanged, CreateCommandPayload, CreateCommandPayloadLog, FB_init, OnCall, ParseResponsePayload, ParseResponsePayloadLog, Reset
        MC_DynamicSpline/
          Structures/
            data type DynamicSplineOutCmd
            data type DynamicSplineParCmd
            data type DynamicSplineRecvData
            data type DynamicSplineSendData
          function block MC_DynamicSplineFB [ST]: CheckFunctionSupported, CheckParameterChanged, CreateCommandPayload, CreateCommandPayloadLog, FB_init, OnCall, ParseResponsePayload, ParseResponsePayloadLog, Reset
        MC_MoveSpline/
          Structures/
            data type MoveSplineOutCmd
            data type MoveSplineParCmd
            data type MoveSplineRecvData
            data type MoveSplineSendData
          function block MC_MoveSplineFB [ST]: CheckFunctionSupported, CheckParameterChanged, CreateCommandPayload, CreateCommandPayloadLog, FB_init, OnCall, ParseResponsePayload, ParseResponsePayloadLog, Reset
      SuperImposing/
        MC_MoveSuperImposed/
          Structures/
            data type MoveSuperImposedOutCmd
            data type MoveSuperImposedParCmd
            data type MoveSuperImposedRecvData
            data type MoveSuperImposedSendData
          function block MC_MoveSuperImposedFB [ST]: CheckFunctionSupported, CheckParameterChanged, CreateCommandPayload, CreateCommandPayloadLog, FB_init, OnCall, ParseResponsePayload, ParseResponsePayloadLog, Reset
        MC_MoveSuperImposedDynamic/
          Structures/
            data type MoveSuperImposedDynamicOutCmd
            data type MoveSuperImposedDynamicParCmd
            data type MoveSuperImposedDynamicRecvData
            data type MoveSuperImposedDynamicSendData
          function block MC_MoveSuperImposedDynamicFB [ST]: CheckFunctionSupported, CheckParameterChanged, CreateCommandPayload, CreateCommandPayloadLog, FB_init, OnCall, ParseResponsePayload, ParseResponsePayloadLog, Reset
      Trigger/
        MC_ReactAtTrigger/
          Structures/
            data type ReactAtTriggerOutCmd
            data type ReactAtTriggerParCmd
            data type ReactAtTriggerRecvData
            data type ReactAtTriggerSendData
          function block MC_ReactAtTriggerFB [ST]: CheckFunctionSupported, CheckParameterChanged, CreateCommandPayload, CreateCommandPayloadLog, FB_init, OnCall, ParseResponsePayload, ParseResponsePayloadLog, Reset
        MC_SetTriggerError/
          Structures/
            data type SetTriggerErrorOutCmd
            data type SetTriggerErrorParCmd
            data type SetTriggerErrorRecvData
            data type SetTriggerErrorSendData
          function block MC_SetTriggerErrorFB [ST]: CheckFunctionSupported, CheckParameterChanged, CreateCommandPayload, CreateCommandPayloadLog, FB_init, OnCall, ParseResponsePayload, ParseResponsePayloadLog, Reset
        MC_SetTriggerLimit/
          Structures/
            data type SetTriggerLimitOutCmd
            data type SetTriggerLimitParCmd
            data type SetTriggerLimitRecvData
            data type SetTriggerLimitSendData
          function block MC_SetTriggerLimitFB [ST]: CheckFunctionSupported, CheckParameterChanged, CreateCommandPayload, CreateCommandPayloadLog, FB_init, OnCall, ParseResponsePayload, ParseResponsePayloadLog, Reset
        MC_SetTriggerMotion/
          Structures/
            data type SetTriggerMotionOutCmd
            data type SetTriggerMotionParCmd
            data type SetTriggerMotionRecvData
            data type SetTriggerMotionSendData
          function block MC_SetTriggerMotionFB [ST]: CheckFunctionSupported, CheckParameterChanged, CreateCommandPayload, CreateCommandPayloadLog, FB_init, OnCall, ParseResponsePayload, ParseResponsePayloadLog, Reset
        MC_SetTriggerRegister/
          Structures/
            data type SetTriggerRegisterOutCmd
            data type SetTriggerRegisterParCmd
            data type SetTriggerRegisterRecvData
            data type SetTriggerRegisterSendData
          function block MC_SetTriggerRegisterFB [ST]: CheckFunctionSupported, CheckParameterChanged, CreateCommandPayload, CreateCommandPayloadLog, FB_init, OnCall, ParseResponsePayload, ParseResponsePayloadLog, Reset
        MC_SetTriggerUser/
          Structures/
            data type SetTriggerUserOutCmd
            data type SetTriggerUserParCmd
            data type SetTriggerUserRecvData
            data type SetTriggerUserSendData
          function block MC_SetTriggerUserFB [ST]: CheckFunctionSupported, CheckParameterChanged, CreateCommandPayload, CreateCommandPayloadLog, FB_init, OnCall, ParseResponsePayload, ParseResponsePayloadLog, Reset
        MC_WaitForTrigger/
          Structures/
            data type WaitForTriggerOutCmd
            data type WaitForTriggerParCmd
            data type WaitForTriggerRecvData
            data type WaitForTriggerSendData
          function block MC_WaitForTriggerFB [ST]: CheckFunctionSupported, CheckParameterChanged, CreateCommandPayload, CreateCommandPayloadLog, FB_init, OnCall, ParseResponsePayload, ParseResponsePayloadLog, Reset
        MC_WaitTime/
          Structures/
            data type WaitTimeOutCmd
            data type WaitTimeParCmd
            data type WaitTimeRecvData
            data type WaitTimeSendData
          function block MC_WaitTimeFB [ST]: CheckFunctionSupported, CheckParameterChanged, CreateCommandPayload, CreateCommandPayloadLog, FB_init, OnCall, ParseResponsePayload, ParseResponsePayloadLog, Reset
      WorkAreas/
        MC_ActivateWorkArea/
          Structures/
            data type ActivateWorkAreaOutCmd
            data type ActivateWorkAreaParCmd
            data type ActivateWorkAreaRecvData
            data type ActivateWorkAreaSendData
          function block MC_ActivateWorkAreaFB [ST]: CheckFunctionSupported, CheckParameterChanged, CreateCommandPayload, CreateCommandPayloadLog, FB_init, OnCall, ParseResponsePayload, ParseResponsePayloadLog, Reset
        MC_MonitorWorkArea/
          Structures/
            data type MonitorWorkAreaOutCmd
            data type MonitorWorkAreaParCmd
            data type MonitorWorkAreaRecvData
            data type MonitorWorkAreaSendData
          function block MC_MonitorWorkAreaFB [ST]: CheckFunctionSupported, CheckParameterChanged, CreateCommandPayload, CreateCommandPayloadLog, FB_init, OnCall, ParseResponsePayload, ParseResponsePayloadLog, Reset
        MC_ReadWorkArea/
          Structures/
            data type ReadWorkAreaOutCmd
            data type ReadWorkAreaParCmd
            data type ReadWorkAreaRecvData
            data type ReadWorkAreaSendData
          function block MC_ReadWorkAreaFB [ST]: CheckFunctionSupported, CheckParameterChanged, CreateCommandPayload, CreateCommandPayloadLog, FB_init, OnCall, ParseResponsePayload, ParseResponsePayloadLog, Reset
        MC_WriteWorkArea/
          Structures/
            data type WriteWorkAreaOutCmd
            data type WriteWorkAreaParCmd
            data type WriteWorkAreaRecvData
            data type WriteWorkAreaSendData
          function block MC_WriteWorkAreaFB [ST]: CheckFunctionSupported, CheckParameterChanged, CreateCommandPayload, CreateCommandPayloadLog, FB_init, OnCall, ParseResponsePayload, ParseResponsePayloadLog, Reset
      Write/
        MC_WriteAnalogOutput/
          Structures/
            data type WriteAnalogOutputOutCmd
            data type WriteAnalogOutputParCmd
            data type WriteAnalogOutputRecvData
            data type WriteAnalogOutputSendData
          function block MC_WriteAnalogOutputFB [ST]: CheckFunctionSupported, CheckParameterChanged, CreateCommandPayload, CreateCommandPayloadLog, FB_init, OnCall, ParseResponsePayload, ParseResponsePayloadLog, Reset
        MC_WriteDigitalOutputs/
          Structures/
            data type WriteDigitalOutputsOutCmd
            data type WriteDigitalOutputsParCmd
            data type WriteDigitalOutputsRecvData
            data type WriteDigitalOutputsSendData
          function block MC_WriteDigitalOutputsFB [ST]: CheckFunctionSupported, CheckParameterChanged, CreateCommandPayload, CreateCommandPayloadLog, FB_init, OnCall, ParseResponsePayload, ParseResponsePayloadLog, Reset
        MC_WriteFrameData/
          Structures/
            data type WriteFrameDataOutCmd
            data type WriteFrameDataParCmd
            data type WriteFrameDataRecvData
            data type WriteFrameDataSendData
          function block MC_WriteFrameDataFB [ST]: CheckFunctionSupported, CheckParameterChanged, CreateCommandPayload, CreateCommandPayloadLog, FB_init, OnCall, ParseResponsePayload, ParseResponsePayloadLog, Reset
        MC_WriteIntegers/
          Structures/
            data type WriteIntegersOutCmd
            data type WriteIntegersParCmd
            data type WriteIntegersRecvData
            data type WriteIntegersSendData
          function block MC_WriteIntegersFB [ST]: CheckFunctionSupported, CheckParameterChanged, CreateCommandPayload, CreateCommandPayloadLog, FB_init, OnCall, ParseResponsePayload, ParseResponsePayloadLog, Reset
        MC_WriteLoadData/
          Structures/
            data type WriteLoadDataOutCmd
            data type WriteLoadDataParCmd
            data type WriteLoadDataRecvData
            data type WriteLoadDataSendData
          function block MC_WriteLoadDataFB [ST]: CheckFunctionSupported, CheckParameterChanged, CreateCommandPayload, CreateCommandPayloadLog, FB_init, OnCall, ParseResponsePayload, ParseResponsePayloadLog, Reset
        MC_WriteReals/
          Structures/
            data type WriteRealsOutCmd
            data type WriteRealsParCmd
            data type WriteRealsRecvData
            data type WriteRealsSendData
          function block MC_WriteRealsFB [ST]: CheckFunctionSupported, CheckParameterChanged, CreateCommandPayload, CreateCommandPayloadLog, FB_init, OnCall, ParseResponsePayload, ParseResponsePayloadLog, Reset
        MC_WriteRobotDefaultDynamics/
          Structures/
            data type WriteRobotDefaultDynamicsOutCmd
            data type WriteRobotDefaultDynamicsParCmd
            data type WriteRobotDefaultDynamicsRecvData
            data type WriteRobotDefaultDynamicsSendData
          function block MC_WriteRobotDefaultDynamicsFB [ST]: CheckFunctionSupported, CheckParameterChanged, CreateCommandPayload, CreateCommandPayloadLog, FB_init, OnCall, ParseResponsePayload, ParseResponsePayloadLog, Reset
        MC_WriteRobotReferenceDynamics/
          Structures/
            data type WriteRobotReferenceDynamicsOutCmd
            data type WriteRobotReferenceDynamicsParCmd
            data type WriteRobotReferenceDynamicsRecvData
            data type WriteRobotReferenceDynamicsSendData
          function block MC_WriteRobotReferenceDynamicsFB [ST]: CheckFunctionSupported, CheckParameterChanged, CreateCommandPayload, CreateCommandPayloadLog, FB_init, OnCall, ParseResponsePayload, ParseResponsePayloadLog, Reset
        MC_WriteRobotSWLimits/
          Structures/
            data type WriteRobotSWLimitsOutCmd
            data type WriteRobotSWLimitsParCmd
            data type WriteRobotSWLimitsRecvData
            data type WriteRobotSWLimitsSendData
          function block MC_WriteRobotSWLimitsFB [ST]: CheckFunctionSupported, CheckParameterChanged, CreateCommandPayload, CreateCommandPayloadLog, FB_init, OnCall, ParseResponsePayload, ParseResponsePayloadLog, Reset
        MC_WriteSystemVariable/
          Structures/
            data type WriteSystemVariableOutCmd
            data type WriteSystemVariableParCmd
            data type WriteSystemVariableRecvData
            data type WriteSystemVariableSendData
          function block MC_WriteSystemVariableFB [ST]: CheckFunctionSupported, CheckParameterChanged, CreateCommandPayload, CreateCommandPayloadLog, FB_init, OnCall, ParseResponsePayload, ParseResponsePayloadLog, Reset
        MC_WriteToolData/
          Structures/
            data type WriteToolDataOutCmd
            data type WriteToolDataParCmd
            data type WriteToolDataRecvData
            data type WriteToolDataSendData
          function block MC_WriteToolDataFB [ST]: CheckFunctionSupported, CheckParameterChanged, CreateCommandPayload, CreateCommandPayloadLog, FB_init, OnCall, ParseResponsePayload, ParseResponsePayloadLog, Reset
    Structures/
      _internal/
        data type SplineDataSend
      AxesGroup/
        Acyclic/
          data type AxesGroupAcyclic
          data type AxesGroupAcyclicAcrEntry
          data type AxesGroupAcyclicAcrEntryCmd
          data type AxesGroupAcyclicAcrEntryCmdBuffer
          data type AxesGroupAcyclicAcrEntryCmdHeader
          data type AxesGroupAcyclicAcrEntryCmdTrigger
          data type AxesGroupAcyclicAcrEntryRsp
          data type AxesGroupAcyclicAcrEntryRspBuffer
          data type AxesGroupAcyclicAcrEntryRspHeader
          data type AxesGroupAcyclicAcrEntryRspTrigger
          data type AxesGroupAcyclicExecutionOrderList
        Cyclic/
          data type AxesGroupCyclic
          data type AxesGroupCyclicPlcToRob
          data type AxesGroupCyclicRobToPlc
        CyclicOptional/
          Internal/
            data type AxesGroupCyclicOptionalDataCartesianPosition
            data type AxesGroupCyclicOptionalDataCartesianPositionExt
            data type AxesGroupCyclicOptionalDataCurrent
            data type AxesGroupCyclicOptionalDataCurrentExt
            data type AxesGroupCyclicOptionalDataForce
            data type AxesGroupCyclicOptionalDataForceExt
            data type AxesGroupCyclicOptionalDataJointPosition
            data type AxesGroupCyclicOptionalDataJointPositionExt
            data type AxesGroupCyclicOptionalDataSubProgram
          data type AxesGroupCyclicOptionalData
          data type AxesGroupCyclicOptionalDataPlcToRob
          data type AxesGroupCyclicOptionalDataRobToPlc
        InternalData/
          data type AxesGroupInternalData
        MessageLog/
          data type AxesGroupMessageLog
        Parameter/
          Cmd/
            data type AxesGroupParameterCmdEntry
          OptionalCyclic/
            data type AxesGroupParameterOptionalCyclic
            data type AxesGroupParameterOptionalCyclicPlcToRob
            data type AxesGroupParameterOptionalCyclicRobToPlc
          Plc/
            data type AxesGroupParameterPlc
            data type AxesGroupParameterPlcOptionalCyclic
            data type AxesGroupParameterPlcParameter
          Rob/
            data type AxesGroupParameterRob
            data type AxesGroupParameterRobOptionalCyclic
            data type AxesGroupParameterRobParameter
          data type AxesGroupParameter
        State/
          DataChanged/
            data type AxesGroupStateDataChanged
          ResetMsg/
            data type AxesGroupStateResetMsg
          RobotData/
            data type AxesGroupRobotData
          Synchronizing/
            data type AxesGroupStateSynchronizing
          SyncState/
            data type AxesGroupStateSyncState
            data type AxesGroupStateSyncStateNo
            data type AxesGroupStateSyncStatePlc
            data type AxesGroupStateSyncStateRob
          data type AxesGroupState
        data type AxesGroup
      Cartesian/
        data type RobotCartesianForce
        data type RobotCartesianForceExt
        data type RobotCartesianForceShort
        data type RobotCartesianPosition
        data type RobotCartesianPositionBase
        data type RobotCartesianPositionExt
        data type RobotCartesianPositionShort
      Common/
        data type CmdHeader
        data type LogParameter
        data type RobotCoordinateSystemParameters
        data type RspHeader
        data type TimeStamp
      Data/
        data type CyclicStateData
        data type FrameData
        data type LoadData
        data type RobotSubProgramData
        data type SplineData
        data type ToolData
        data type UserData
      DatenAndTime/
        data type IEC_DATE
        data type IEC_TIME
        data type IEC_TIMESTAMP
        data type SystemTime
      Dynamics/
        data type DefaultDynamics
        data type ReferenceDynamics
      Joint/
        data type RobotJointCurrent
        data type RobotJointCurrentExt
        data type RobotJointCurrentShort
        data type RobotJointPosition
        data type RobotJointPositionExt
        data type RobotJointPositionShort
      Miscellaneous/
        data type AlarmMessage
        data type ArmConfigParameter
        data type AuxOffset
        data type CoordinateSystem
        data type DataEnableSync
        data type DataInSync
        data type DHParameter
        data type ExternalAxesFlags
        data type ForceStatus
        data type FragmentAction
        data type JogControl
        data type MeasuringInputResult
        data type ProcessingModeAllowed
        data type RaStatusWord
        data type RCSupportedFunctions
        data type RobotAxesFlags
        data type SWLimits
        data type SynchronizationModes
        data type TrackingStatus
        data type TurnNumber
        data type VersionStruct
      Telegram/
        Common/
        PlcToRob/
          Command/
            data type TelegramPlcToRobCommand
            data type TelegramPlcToRobCommandHeader
          Cyclic/
            data type TelegramPlcToRobCyclicData
          CyclicOptional/
            Internal/
              data type TelegramPlcToRobCyclicOptionalCartesianPosition
              data type TelegramPlcToRobCyclicOptionalCartesianPositionExt
              data type TelegramPlcToRobCyclicOptionalCurrent
              data type TelegramPlcToRobCyclicOptionalCurrentExt
              data type TelegramPlcToRobCyclicOptionalForce
              data type TelegramPlcToRobCyclicOptionalForceExt
              data type TelegramPlcToRobCyclicOptionalJointPosition
              data type TelegramPlcToRobCyclicOptionalJointPositionExt
              data type TelegramPlcToRobCyclicOptionalSubProgramData
            data type TelegramPlcToRobCyclicOptionalData
          Footer/
            data type TelegramPlcToRobFooter
          Fragment/
            data type TelegramPlcToRobFragment
            data type TelegramPlcToRobFragmentHeader
          Header/
            data type TelegramPlcToRobHeader
          Sequence/
            data type TelegramPlcToRobSequence
            data type TelegramPlcToRobSequenceHeader
          data type TelegramPlcToRob
        RobToPlc/
          Command/
            data type TelegramRobToPlcCommand
            data type TelegramRobToPlcCommandHeader
          CyclicOptional/
            Internal/
              data type TelegramRobToPlcCyclicOptionalCartesianPosition
              data type TelegramRobToPlcCyclicOptionalCartesianPositionExt
              data type TelegramRobToPlcCyclicOptionalCurrent
              data type TelegramRobToPlcCyclicOptionalCurrentExt
              data type TelegramRobToPlcCyclicOptionalForce
              data type TelegramRobToPlcCyclicOptionalForceExt
              data type TelegramRobToPlcCyclicOptionalJointPosition
              data type TelegramRobToPlcCyclicOptionalJointPositionExt
              data type TelegramRobToPlcCyclicOptionalSubProgramData
            data type TelegramRobToPlcCyclicOptionalData
          Footer/
            data type TelegramRobToPlcFooter
          Fragment/
            data type TelegramRobToPlcFragment
            data type TelegramRobToPlcFragmentHeader
          Header/
            data type TelegramRobToPlcHeader
          Sequence/
            data type TelegramRobToPlcSequence
            data type TelegramRobToPlcSequenceHeader
          data type TelegramRobToPlc
        data type Telegram
      WorkArea/
        data type RobotWorkArea
        data type RobotWorkAreaLimitCartesian
        data type RobotWorkAreaLimitJoint
      data type ExecutionModeAllowed
      data type MessageHeaderCommand
      data type MessageHeaderResponse
*)

// Library/Enumerations/ArmConfig/ArmConfigElbow
{attribute 'qualified_only'}
// ------------------------------------------------------------------------- 
//  SRCI Robot Library                                                
// ------------------------------------------------------------------------- 
//                                                                           
//  Object:      ArmConfigElbow                                       
//  Author:      Thorsten Brach                                                
//  Date:        2024-06-01
//
//  Description:                                              
//   
//                                                                           
//  Copyright: 
//    (C) 2024 Thorsten Brach. All rights reserved                                                                                                                                            
//             Licensed under the LGPL-3.0 license.
//                                                                           
//  Disclaimer:                                                                           
//    This project is provided without any guarantee and can be used for   
//    private and commercial purposes. Any use is at the user’s 
//    own risk and responsibility.
//
// -------------------------------------------------------------------------
TYPE ArmConfigElbow :
(
 /// Use config in position  
 USE_CONFIG := 0,
 /// Do not change config with this movement. (default)
 SAME := 1,
 /// Configuration in position is not used but the Robot is free to change config
 FREE := 2,
 /// Set elbow configuration in position to Down
 DOWN := 3,
 /// Set elbow configuration in position to up
 UP := 4
);
END_TYPE

// Library/Enumerations/ArmConfig/ArmConfigShoulder
{attribute 'qualified_only'}
// ------------------------------------------------------------------------- 
//  SRCI Robot Library                                                
// ------------------------------------------------------------------------- 
//                                                                           
//  Object:      ArmConfigShoulder                                       
//  Author:      Thorsten Brach                                                
//  Date:        2024-06-01
//
//  Description:                                              
//   
//                                                                           
//  Copyright: 
//    (C) 2024 Thorsten Brach. All rights reserved                                                                                                                                            
//             Licensed under the LGPL-3.0 license.
//                                                                           
//  Disclaimer:                                                                           
//    This project is provided without any guarantee and can be used for   
//    private and commercial purposes. Any use is at the user’s 
//    own risk and responsibility.
//
// -------------------------------------------------------------------------
TYPE ArmConfigShoulder :
(
 /// Use config in position  
 USE_CONFIG := 0,
 /// Do not change config with this movement. (default)
 SAME := 1,
 /// Configuration in position is not used but the Robot is free to change config
 FREE := 2,
 /// Set shoulder configuration in position to Back
 BACK := 3,
 /// Set shoulder configuration in position to Front
 FRONT := 4
);
END_TYPE

// Library/Enumerations/ArmConfig/ArmConfigWrist
{attribute 'qualified_only'}
// ------------------------------------------------------------------------- 
//  SRCI Robot Library                                                
// ------------------------------------------------------------------------- 
//                                                                           
//  Object:      ArmConfigWrist                                       
//  Author:      Thorsten Brach                                                
//  Date:        2024-06-01
//
//  Description:                                              
//   
//                                                                           
//  Copyright: 
//    (C) 2024 Thorsten Brach. All rights reserved                                                                                                                                            
//             Licensed under the LGPL-3.0 license.
//                                                                           
//  Disclaimer:                                                                           
//    This project is provided without any guarantee and can be used for   
//    private and commercial purposes. Any use is at the user’s 
//    own risk and responsibility.
//
// -------------------------------------------------------------------------
TYPE ArmConfigWrist :
(
 /// Use config in position  
 USE_CONFIG := 0,
 /// Do not change config with this movement. (default)
 SAME := 1,
 /// Configuration in position is not used but the Robot is free to change config
 FREE := 2,
 /// Set wrist configuration in position to Flip
 FLIP := 3,
 /// Set wrist configuration in position to Non-Flip
 NON_FLIP := 4
);
END_TYPE

// Library/Enumerations/Events/RobotLibraryErrorIdEnum
{attribute 'qualified_only'}
TYPE RobotLibraryErrorIdEnum :
(
  NO_ERROR := 0,

  /// Telegram control does not match the telegram state
  ERR_TELEGRAM_CONTROL_MISMATCH_TELEGRAM_STATE_0xA1 := 16#A1,  
  /// Initialization lost for unknown reason. See message log after reinitializing
  ERR_INIT_LOST_UNKNOWN_0xA2  := 16#A2,
  /// Telegram length does not match the length provided in the communication interface.
  ERR_TELEGRAM_LENGTH_MISMATCH_0xA3 := 16#A3,
  /// Incompatible major SRCI version
  ERR_SRCI_MAJOR_VERSION_INCOMPATIBLE_0xA4 := 16#A4,
  /// Lifesign timeout
  ERR_LIFESIGN_TIMEOUT_0xA5 := 16#A5,
  /// The selected optional cyclic data does not fit in the given telegram size
  ERR_CYCLIC_DATA_TOO_LARGE_0xA6 := 16#A6,
  /// The robot interface was reset after being initialized
  ERR_INTERFACE_WAS_RESET_AFTER_INIT_0xA7 := 16#A7,
  /// Telegram sequence timeout
  ERR_TELEGRAM_SEQ_TIMEOUT_0xA8 := 16#A8,
  /// The telegram number changed after initialization
  ERR_TELEGRAM_NO_CHANGED_AFTER_INIT_0xA9 := 16#A9,
  /// Invalid AxesGroupID
  ERR_AXESGROUP_ID_INVALID_0xAA := 16#AA,
  /// Telegram number is invalid. E.g. TwoSequences is only activated in one direction
  ERR_TELEGRAM_NUMBER_INVALID_0xAB := 16#AB,
  /// Telegram Number is not supported
  ERR_TELEGRAM_NUMBER_NOT_SUPPORTED_0xAC := 16#AC,
  /// Server Connection to the communication partner was lost
  ERR_SERVER_CONNECTION_LOST_0xAD := 16#AD,
  
  
  /// Table 5-96: Telegram and Initialization State 
  /// Initialization may fail due to several reasons, described in the following table. T he failure is
  /// signaled using the telegram state byte.
 

  /// 7.1 Table "A" – Command ErrorIDs 
  /// If an error related to the execution of a function block occurs, the function block returns an ErrorID
  /// to specify the error. The errors are stored in the PLC message buffer and are displayed on the
  /// function block outputs.
  /// In the PLC message buffer, they are dynamically arranged by the client to be displayed as follows:
  /// <Origin> <MessageType> <Command name> <Description>
  /// More information about the general message handling mechanism can be found in 5.5.11
  /// Diagnostics.
  /// The following table gives an overview over the existing ErrorIDs reported by commands and the
  /// corresponding description.

  /// ------------------------------------------------------
  /// CLIENT ErrorIDs
  /// ------------------------------------------------------

  /// Client Specified Velocity not valid
  /// Commands using the parameter "Velocity"
  ERR_VELOCITY_INVALID  := 16#8401,
  
  /// Client Specified Acceleration not valid
  /// Commands using the parameter "Acceleration"
  ERR_ACCELERATION_INVALID  := 16#8402,
  
  /// Client Specified Deceleration not valid
  /// Commands using the parameter "Deceleration"
  ERR_DECELERATION_INVALID  := 16#8403,
  
  /// Client Specified Jerk not valid
  /// Commands using the parameter "Jerk"
  ERR_JERK_INVALID  := 16#8404,
  
  /// Client Invalid parameter value - ConfigMode Elbow
  /// Commands using the parameter "ConfigMode"
  ERR_CONFIGMODE_ELBOW_INVALID  := 16#8405,
  
  /// Client Invalid parameter value - ConfigMode Shoulder
  /// Commands using the parameter "ConfigMode"
  ERR_CONFIGMODE_SHOULDER_INVALID  := 16#8406,
  
  /// Client Invalid parameter value - ConfigMode Wrist
  /// Commands using the parameter "ConfigMode"
  ERR_CONFIGMODE_WRIST_INVALID  := 16#8407,
  
  /// Client Invalid parameter value - TrajectoryMode
  /// Commands using the parameter "TrajectoryMode"
  ERR_TRAJECTORYMODE_INVALID  := 16#8409,
  
  /// Client Invalid parameter value - Override
  /// Commands using the parameter "Override"
  ERR_OVERRIDE_INVALID  := 16#8410,
  
  /// Client Invalid parameter value - AbortingMode.
  /// Only 0: Buffer / 1: Abort are valid.
  /// Commands using the parameter "AbortingMode"
  ERR_ABORTINGMODE_INVALID  := 16#8411,
  
  /// Client Invalid parameter value - ToolNo outside of
  /// the allowed range -1..254
  /// Commands using the parameter "ToolNo"
  ERR_TOOLNO_RANGE  := 16#8412,
  
  /// Client Invalid parameter value - ToolNo not
  /// available on RC
  /// Commands using the parameter "ToolNo"
  ERR_TOOLNO_UNAVAILABLE  := 16#8413,
  
  /// Client Invalid parameter value - FrameNo outside
  /// of the allowed range -1..254
  /// Commands using the parameter "FrameNo"
  ERR_FRAMENO_RANGE  := 16#8414,
  
  /// Client Invalid parameter value - FrameNo not
  /// available on RC
  /// Commands using the parameter "FrameNo"
  ERR_FRAMENO_UNAVAILABLE  := 16#8415,
  
  /// Client The array specified for AcyclicData exceeds
  /// the supported maximum length of 190 bytes
  /// Command "CallSubprogram"
  ERR_ACYCLICDATA_TOO_LARGE  := 16#8416,
  
  /// Client The array length specified for ReturnAcyclicData
  /// is not sufficient for the returned data. The data has been truncated
  /// Command "CallSubprogram"
  ERR_RETURNACYCLICDATA_TRUNCATED  := 16#8417,
  
  /// Client Invalid parameter value - LoadNo outside of
  /// the allowed range -1..254
  /// All commands
  ERR_LOADNO_RANGE  := 16#8418,
  
  /// Client Specified ProcessingMode not defined
  /// Commands using the parameter "ProcessingMode"
  ERR_PROCESSINGMODE_NOT_DEFINED  := 16#8602,
  
  /// Client Specified ProcessingMode not allowed
  /// Commands using the parameter "ProcessingMode"
  ERR_PROCESSINGMODE_NOT_ALLOWED  := 16#8603,
  
  /// Client Specified Emitter ID not allowed
  /// Commands using the parameter "EmitterID"
  ERR_EMITTERID_NOT_ALLOWED := 16#8604,
  
  /// Client Specified Listener ID not allowed
  /// Commands using the parameter "ListenerID"
  ERR_LISTENERID_NOT_ALLOWED   := 16#8605,
  
  /// Client ProcessingMode or SequenceFlag changed during execution
  /// Commands using the parameter "ProcessingMode" or "SequenceFlag"
  ERR_PROCSEQFLAG_CHANGED  := 16#8609,
  
  /// Client Commands are not Enabled (First Robot must be initialized)
  /// All commands
  ERR_COMMANDS_NOT_ENABLED  := 16#8612,
  
  /// Client Error received from robot without error ID
  /// All commands
  ERR_ROBOT_ERROR_NO_ID  := 16#8613,
  
  /// Client AxesGroup changed during execution
  /// All commands
  ERR_AXESGROUP_CHANGED  := 16#8614,
  
  /// Client Specified SEQ Flag not allowed
  /// Commands using the parameter "SequenceFlag"
  ERR_SEQFLAG_NOT_ALLOWED  := 16#8616,
  
  /// Client AxesGroup cleared during execution
  /// All commands
  ERR_AXESGROUP_CLEARED  := 16#8617,
  
  /// Client No free ACR entry available
  /// All commands
  ERR_NO_FREE_ACR_ENTRY  := 16#8618,
  
  /// Client Sequence flag must be 0 in the selected ProcessingMode
  /// Commands using the parameter "ProcessingMode" or "SequenceFlag"
  ERR_SEQFLAG_INVALID_IN_PROC_MODE  := 16#8625,
  
  /// Client Specified Listener ID must be > 0 for selected trigger based ProcessingMode
  /// Commands using the parameter "ListenerID"
  ERR_LISTENERID_MUST_BE_GREATER_THAN_ZERO  := 16#8626,
  
  /// Client Specified Emitter ID must be 0
  /// Commands using the parameter "EmitterID"
  ERR_EMITTERID_MUST_BE_ZERO  := 16#8627,
  
  /// Client Specified Listener ID must be a positive value (>= 0)
  /// Commands using the parameter "ListenerID"
  ERR_LISTENERID_MUST_BE_POSITIVE  := 16#8635,


  /// ------------------------------------------------------
  /// SERVER ErrorIDs
  /// ------------------------------------------------------
  
  /// Server Continue not possible - robot is not enabled
  /// Command "GroupContinue"
  ERROR_CONTINUE_NOT_POSSIBLE_BY_NOT_ENABLED := 16#8C01,
  
  /// Server Continue not possible - robot is not inPrimaryPosition
  /// Command "GroupContinue"
  ERROR_CONTINUE_NOT_POSSIBLE_BY_NOT_IN_PRIMARY_POS := 16#8C02,
  
  /// Server Robot disabled
  /// Command "EnableRobot"
  ERR_ROBOT_DISABLED  := 16#8C03,
  /// Server Robot disabled due to an error
  /// Command "EnableRobot"
  ERR_ROBOT_DISABLED_BY_ERROR  := 16#8C04,

  /// Server Not all mandatory commands have been called yet
  /// Command "EnableRobot"
  ERR_MANDATORY_CMDS_MISSING  := 16#8C05,

  /// Server RI state is NOT_SYNCHRONIZED and the respective syncReaction denies enabling in this state
  /// Command "EnableRobot"
  ERR_RI_NOT_SYNCHRONIZED  := 16#8C06,

  /// Server Limit exceeded. Move closer to return position
  /// Command "ReturnToPrimary"
  ERR_LIMIT_EXCEEDED_RETURN_POS  := 16#8C07,

  /// Server Invalid parameter value - Must switch to T1Ext when changing between AutoExt and T2Ext
  /// Command "SetOperationMode"
  ERR_SET_OPMODE_T1EXT_REQUIRED  := 16#8C08,

  /// Server Cannot write to a dynamic frame (frame used by e.g. conveyor tracking)
  /// Command "WriteFrameData"
  ERR_WRITE_DYNAMIC_FRAME  := 16#8C09,

  /// Server Continue not possible in manual operation mode
  /// Command "GroupContinue"
  ERR_CONTINUE_NOT_POSSIBLE_BY_MANUAL_MODE  := 16#8C10,

  /// Server It is not allowed to reference a frame which already references another frame
  /// Command "WriteFrame"
  ERR_FRAME_REFERENCING_INVALID  := 16#8C12,

  /// Server The referenced Frame is invalid, dynamic (frame used by e.g. conveyor tracking) or does not exist
  /// Command "WriteFrame"
  ERR_FRAME_INVALID  := 16#8C13,

  /// Server Currently used tool ID differs from the tool ID of the target position
  /// Command "ReturnToPrimary"
  ERR_TOOLID_DIFFERS_TARGET  := 16#8C14,

  /// Server Writing a Frame during an active movement is not supported by this RC
  /// Command "WriteFrame"
  ERR_WRITE_FRAME_DURING_MOVE  := 16#8C15,

  /// Server Writing a Tool during an active movement is not supported by this RC
  /// Command "WriteToolData"
  ERR_WRITE_TOOL_DURING_MOVE  := 16#8C16,

  /// Server Writing a Load during an active movement is not supported by this RC
  /// Command "WriteLoadData"
  ERR_WRITE_LOAD_DURING_MOVE  := 16#8C17,

  /// Server ManualStep is not allowed in Automatic External
  /// Command "EnableRobot"
  ERR_MANUAL_STEP_NOT_ALLOWED  := 16#8C20,

  /// Server ManualStep is only allowed when StepMode is active
  /// Command "EnableRobot"
  ERR_MANUAL_STEP_ONLY_IN_STEP_MODE_ALLOWED  := 16#8C21,

  /// Server The current ToolData has changed and differs from the one when the primary position was left. Returning is not possible.
  /// Command "ReturnToPrimary"
  ERR_TOOLDATA_DIFFERS  := 16#8C22,

  /// Server The current LoadData has changed and differs from the one when the primary position was left. Returning is not possible.
  /// Command "ReturnToPrimary"
  ERR_LOADDATA_DIFFERS := 16#8C23,

  /// Server The current FrameData has changed and differs from the one when the primary position was left. Returning is not possible.
  /// Command "ReturnToPrimary"
  ERR_FRAMEDATA_DIFFERS := 16#8C24,

  /// Server The current reference FrameData has changed and differs from the one when the primary position was left. Returning is not possible.
  /// Command "ReturnToPrimary"
  ERR_REF_FRAMEDATA_CHANGED  := 16#8C25,

  /// Server The ToolNo differs from the one in the return position. Returning is not possible.
  /// Command "ReturnToPrimary"
  ERR_TOOLNO_DIFFERS_TARGET  := 16#8C26,

  /// Server The FrameNo differs from the one in the return position. Returning is not possible.
  /// Command "ReturnToPrimary"
  ERR_FRAMENO_DIFFERS_TARGET  := 16#8C27,

  /// Server Continue is not possible while the Robot is interrupting or stopping.
  /// Command "GroupContinue"
  ERR_CONTINUE_WHILE_STOPPING  := 16#8C28,

  /// Server Software limits could not be set because values were specified for non-existing axes
  /// Command "WriteSWLimits"
  ERR_SOFTWARE_LIMITS_FOR_NON_EXISTING_AXIS  := 16#8C29,

  /// Server RI state is NOT_SYNCHRONIZED and the respective syncReaction denies continue in this state
  /// Command "GroupContinue"
  ERR_RI_NOT_SYNCHRONIZED_CONTINUE_DENIED  := 16#8C30,

  /// Server Enable switch must be active to enable the robot
  /// Command "EnableRobot"
  ERR_ENABLE_SWITCH_REQUIRED  := 16#8C31,

  /// Server Manual step sent while robot not enabled
  /// Command "EnableRobot"
  ERR_MANUAL_STEP_WHILE_DISABLED  := 16#8C32,

  /// Server Jog not possible during active movement
  /// Command "GroupJog"
  ERR_JOG_NOT_ALLOWED_DURING_MOVE  := 16#8C33,

  /// Server Target position was commanded for an external axis which does not exist
  /// All move commands
  ERR_TARGET_POS_FOR_NON_EXISTING_AXIS  := 16#8C34,

  /// Server Jog of axis is not possible. Axis does not exist
  /// Command "GroupJog"
  ERR_JOG_AXIS_NOT_EXIST  := 16#8C35,

  /// Server Incremental jog is only possible in one axis of rotation
  /// Command "GroupJog"
  ERR_INC_JOG_ONE_AXIS_ONLY  := 16#8C36,

  /// Server A program for the supplied JobID does not exist.
  /// Commands: "CallSubprogram", "StopSubprogram"
  ERR_JOBID_NOT_EXIST  := 16#8C37,

  /// Server A program including motion commands is only allowed to be executed in a sequence buffer
  /// Command "CallSubprogram"
  ERR_ONLY_ALLOWED_IN_SEQ_BUFFER  := 16#8C38,

  /// Server A program with the same number is already running. Multiple instances are not supported
  /// Command "CallSubprogram"
  ERR_JOB_ALREADY_RUNNING  := 16#8C39,

  /// Server Changing the JobID in PM 3 during runtime of this CMD is not supported.
  /// Command "CallSubprogram"
  ERR_JOBID_CHANGE_PM3_NOT_ALLOWED  := 16#8C42,

  /// Server Continue is not possible while the robot is stopping due to GroupInterrupt, GroupStop, SetSequence, or GroupJog
  /// Command "GroupContinue"
  ERR_CONTINUE_DURING_STOPPING  := 16#8C43,

  /// Server GroupJog motion was stopped due to the release of the enable switch.
  /// Command "GroupJog"
  ERR_JOG_STOPPED_BY_ENABLE_RELEASED  := 16#8C52,

  /// Server Setting the limits is not possible because the current robot position is currently outside of those limits.
  /// Command "WriteSWLimits"
  ERR_SWLIMITS_NOT_ALLOWED_ROBOT_IS_OUTSIDE  := 16#8C53,

  /// Server Setting the limits is not possible while a motion is active.
  /// Command "WriteSWLimits"
  ERR_SWLIMITS_NOT_ALLOWED_DURING_MOVE  := 16#8C54,

  /// Server Change of operation mode by the PLC not possible. The RC must be in an "External" operation mode
  /// Command "SetOperationMode"
  ERR_OPMODE_CHANGE_NOT_POSSIBLE_BY_PLC  := 16#8C56,

  /// Server Auxpoint must not be identical to start or end position of the motion
  /// Commands: "MoveCircularAbsolute", "MoveCircularRelative", "MoveCircularCam"
  ERR_AUXPOINT_IDENTICAL_WITH_OTHER_POS  := 16#8C57,

  /// Server Auxpoint invalid
  /// Commands: "MoveCircularAbsolute", "MoveCircularRelative", "MoveCircularCam"
  ERR_AUXPOINT_INVALID  := 16#8C58,

  /// Server Supplied positions must not be identical or at a larger distance apart
  /// Commands: "CalculateTool", "CalculateFrame"
  ERR_CALC_NOT_POSSIBLE_BY_POS := 16#8C59,

  /// Server Calculation not possible with the given parameters
  /// Commands: "CalculateTool", "CalculateFrame"
  ERR_CALC_NOT_POSSIBLE_BY_PARA  := 16#8C60,

  /// Server Positions must not be on one line
  /// Commands: "CalculateTool", "CalculateFrame"
  ERR_CALC_NOT_POSSIBLE_BY_POS_ON_LINE := 16#8C61,

  /// Server No solution found for the given CartesianPosition
  /// Command "CalculateInverseKinematic"
  ERR_INV_KINEMATIC_NO_SOLUTION := 16#8C62,

  /// Server Solution is outside of the hardware limits
  /// Commands: "CalculateInverseKinematic", "CalculateForwardKinematic"
  ERR_INV_KINEMATIC_SOLUTION_OUTSIDE_SWLIMITS := 16#8C63,

  /// Server The selected parameter is write protected and can thus not be changed
  /// Command "WriteSystemVariable"
  ERR_PARAM_WRITE_PROTECTED  := 16#8C64,

  /// Server Number of received positions exceeds the maximum expected number (index out of range)
  /// Commands: "CalculateTool", "CalculateFrame"
  ERR_POS_INDEX_OUT_OF_RANGE  := 16#8C65,

  /// Server Number of received positions does not correspond to the required number for the selected mode
  /// Commands: "CalculateTool", "CalculateFrame"
  ERR_POS_INDEX_MISMATCH  := 16#8C66,

  /// Server Invalid parameter value - AccelerationRate
  /// Commands using the parameter "AccelerationRate"
  ERR_INVALID_PARAM_ACCELERATION_RATE := 16#8D01,

  /// Server Invalid parameter value - BlendingMode
  /// Commands using the parameter "BlendingMode"
  ERR_INVALID_PARAM_BLENDING_MODE := 16#8D03,

  /// Server Invalid parameter value - BlendingParameter
  /// Commands using the parameter "BlendingParameter"
  ERR_INVALID_PARAM_BLENDING_PARA  := 16#8D04,

  /// Server Invalid parameter value - ConfigMode Elbow
  /// Commands using the parameter "ConfigMode"
  ERR_INVALID_PARAM_CONFIGMODE_ELBOW := 16#8D05,

  /// Server Invalid parameter value - DecelerationRate
  /// Commands using the parameter "DecelerationRate"
  ERR_INVALID_PARAM_DECELERATION_RATE := 16#8D06,

  /// Server Invalid parameter value - No value greater than zero
  /// Commands: "WriteDefaultDynamics", "WriteReferenceDynamics"
  ERR_INVALID_PARAM_VALUE_ZERO := 16#8D07,

  /// Server Invalid parameter value - FrameNo
  /// Commands using the parameter "FrameNo"
  ERR_INVALID_PARAM_FRAMENO := 16#8D08,

  /// Server Invalid parameter value - IncrementalRotation
  /// Command "GroupJog"
  ERR_INVALID_PARAM_INC_ROTATION  := 16#8D09,

  /// Server Invalid parameter value - IncrementalTranslation
  /// Command "GroupJog"
  ERR_INVALID_PARAM_INC_TRANSLATION := 16#8D10,

  /// Server Invalid parameter value - JerkRate
  /// Commands using the parameter "JerkRate"
  ERR_INVALID_PARAM_JERK_RATE := 16#8D11,

  /// Server Invalid parameter value - Control Positive and negative jog direction was active at the same time
  /// Command "GroupJog"
  ERR_INVALID_PARAM_JOG_POS_AND_JOG_NEG := 16#8D12,

  /// Server Invalid parameter value - JointPosition
  /// Commands using the parameter "JointPosition"
  ERR_INVALID_PARAM_JOINT_POS := 16#8D13,

  /// Server Invalid parameter value - LifesignTimeout
  /// Command "ExchangeConfiguration"
  ERR_INVALID_PARAM_LIFE_SIGN_TIMEOUT := 16#8D14,

  /// Server Invalid parameter value - SoftwareLimits all values must not be zero
  /// Command "WriteRobotSWLimits"
  ERR_INVALID_PARAM_SWLIMITS := 16#8D15,

  /// Server Invalid parameter value - LimitValues
  /// Command "WriteRobotSWLimits"
  ERR_INVALID_PARAM_LIMITVALUES := 16#8D16,

  /// Server Invalid parameter value - LoadNo
  /// Commands using the parameter "LoadNo"
  ERR_INVALID_PARAM_LOADNO := 16#8D17,

  /// Server Invalid parameter value - LogLevel
  /// Command "ExchangeConfiguration"
  ERR_INVALID_PARAM_LOG_LEVEL := 16#8D18,

  /// Server Invalid parameter value - Mode
  /// Commands using the parameter "Mode"
  ERR_INVALID_PARAM_MODE := 16#8D21,

  /// Server Invalid parameter value - OriMode
  /// Commands using the parameter "OriMode"
  ERR_INVALID_PARAM_ORI_MODE := 16#8D22,

  /// Server Invalid parameter value - Override
  /// Commands using the parameter "Override"
  ERR_INVALID_PARAM_OVERRIDE := 16#8D23,

  /// Server Invalid parameter value - Position
  /// Commands using the parameter "Position"
  ERR_INVALID_PARAM_POSITION := 16#8D24,

  /// Server Invalid parameter value - ReferenceDynamics all values less than zero
  /// Command "WriteReferenceDynamics"
  ERR_INVALID_PARAM_REF_DYNAMICS_LESS_THAN_ZERO := 16#8D25,

  /// Server Invalid parameter value - Acceleration
  /// Commands using the parameter "Acceleration"
  ERR_INVALID_PARAM_ACCELERATION := 16#8D26,

  /// Server Invalid parameter value - Deceleration
  /// Commands using the parameter "Deceleration"
  ERR_INVALID_PARAM_DECELERATION := 16#8D27,

  /// Server Invalid parameter value - Jerk
  /// Commands using the parameter "Jerk"
  ERR_INVALID_PARAM_JERK := 16#8D28,

  /// Server Invalid parameter value - Velocity
  /// Commands using the parameter "Velocity"
  ERR_INVALID_PARAM_VELOCITY := 16#8D29,

  /// Server Invalid parameter value - ReturnMode
  /// Command "ReturnToPrimary"
  ERR_INVALID_PARAM_RETURN_MODE := 16#8D30,

  /// Server Invalid parameter value - TargetSequence
  /// Command "SetSequence"
  ERR_INVALID_PARAM_TARGET_SEQUENCE := 16#8D31,

  /// Server Invalid parameter value - OperationMode
  /// Command "SetOperationMode"
  ERR_INVALID_PARAM_OPERATION_MODE := 16#8D32,

  /// Server Invalid parameter value - SyncReaction
  /// Command "LRob_ExchangeConfiguration"
  ERR_INVALID_PARAM_SYNC_REACTION := 16#8D33,

  /// Server Invalid parameter value - Time
  /// Commands using the parameter "Time"
  ERR_INVALID_PARAM_TIME := 16#8D34,

  /// Server Invalid parameter value - ToolNo
  /// Commands using the parameter "ToolNo"
  ERR_INVALID_PARAM_TOOLNO := 16#8D35,

  /// Server Invalid parameter value - TrajectoryMode
  /// Command "ReturnToPrimary"
  ERR_INVALID_PARAM_TRAJECTORY_MODE := 16#8D36,

  /// Server Invalid parameter value - TurnMode
  /// Commands using the parameter "TurnMode"
  ERR_INVALID_PARAM_TURN_MODE := 16#8D37,

  /// Server Invalid parameter value - VelocityRate
  /// Commands using the parameter "VelocityRate"
  ERR_INVALID_PARAM_VELOCITY_MODE := 16#8D38,

  /// Server Invalid parameter value - WaitForNrOfCmd
  /// Command "LRob_ExchangeConfiguration"
  ERR_INVALID_PARAM_WAIT_FOR_NR_OF_CMD := 16#8D39,

  /// Server Invalid parameter value - ConfigMode Shoulder
  /// Commands using the parameter "ConfigMode"
  ERR_INVALID_PARAM_CONFIG_MODE_SHOULDER := 16#8D40,

  /// Server Invalid parameter value - ConfigMode Wrist
  /// Commands using the parameter "ConfigMode"
  ERR_INVALID_PARAM_CONFIG_MODE_WRIST := 16#8D41,

  /// Server Invalid parameter value - StepMode
  /// Commands using the parameter "StepMode"
  ERR_INVALID_PARAM_STEP_MODE := 16#8D42,

  /// Server The supplied StopMode is not valid. Use 0, 1, or 2
  /// Command "StopSubprogram"
  ERR_STEP_MODE_NOT_VALID := 16#8D43,

  /// Server When StopMode 2: (Stop all subprograms) is selected, the TargetID must be -1.
  /// Command "StopSubprogram"
  ERR_STOP_MODE_2_TARGETID_NEG1 := 16#8D44,

  /// Server When StopMode 0: (Stop via JobID) is selected, the TargetID must NOT be -1.
  /// Command "StopSubprogram"
  ERR_STOP_MODE_0_TARGETID_NOT_NEG1 := 16#8D45,

  /// Server When StopMode 1: (Stop via InstanceID) is selected, the TargetID must NOT be -1.
  /// Command "StopSubprogram"
  ERR_STOP_MODE_1_TARGETID_NOT_NEG1  := 16#8D46,

  /// Server Invalid parameter value - Index out of range
  /// All Commands
  ERR_INVALID_PARAM_INDEX_OUT_OF_RANGE := 16#8D47,

  /// Server Invalid parameter value - Same index was used multiple times
  /// Commands: "WriteDigitalOutputs", "WriteIntegers", "WriteReals", "WriteAnalogOutputs", "ReadDigitalInputs", "ReadDigitalOutputs", "ReadIntegers", "ReadReals"
  ERR_INVALID_PARAM_SAME_INDEX_MULTIPLE_TIMES := 16#8D48,

  /// Server Invalid parameter value - Specified mass greater than the maximum RA payload.
  /// Command "WriteLoad"
  ERR_INVALID_PARAM_MASS_EXCEEDS_PAYLOAD  := 16#8D49,

  /// Server Invalid parameter value - At least one index must not be 0 and result in a read/write operation.
  /// Commands: "WriteDigitalOutputs", "WriteIntegers", "WriteReals", "WriteAnalogOutputs", "ReadDigitalInputs", "ReadDigitalOutputs", "ReadIntegers", "ReadReals"
  ERR_INVALID_PARAM_AT_LEAST_ONE_INDEX_REQUIRED  := 16#8D50,

  /// Server Invalid parameter value - MessageLevel must be between 0-28
  /// Command "ReadMessages"
  ERR_INVALID_PARAM_MESSAGE_LEVEL := 16#8D51,

  /// Server Invalid parameter value - CircPlane does not match CircMode
  /// Commands: "MoveCircularAbsolute", "MoveCircularRelative", "MoveCircularCam"
  ERR_INVALID_PARAM_CIRCPLANE_MISMATCH_CIRCMODE := 16#8D61,

  /// Server Invalid parameter value - CircMode outside of the allowed range 0..3
  /// Commands: "MoveCircularAbsolute", "MoveCircularRelative", "MoveCircularCam"
  ERR_INVALID_PARAM_CIRCMODE_OUT_OF_RANGE := 16#8D62,

  /// Server Invalid parameter value - Tolerance must only be used for CircMode 1
  /// Commands: "MoveCircularAbsolute", "MoveCircularRelative", "MoveCircularCam"
  ERR_INVALID_PARAM_TOLERANCE_ONLY_CIRCMODE_1 := 16#8D63,

  /// Server Invalid parameter value - Angle must only be used for CircMode 2
  /// Commands: "MoveCircularAbsolute", "MoveCircularRelative", "MoveCircularCam"
  ERR_INVALID_PARAM_ANGLE_ONLY_CIRCMODE_2 := 16#8D64,

  /// Server Invalid parameter value - PathChoice outside of the allowed range 0..1
  /// Commands
  ERR_INVALID_PARAM_PATH_CHOICE_OUT_OF_RANGE := 16#8D65,

  /// Server Invalid parameter value - Mode outside of the allowed range 0..4
  /// Command "ShiftPosition"
  ERR_INVALID_PARAM_SHIFT_MODE_OUT_OF_RANGE := 16#8D66,

  /// Server Invalid parameter value - RotationAngle only allowed in mode 3
  /// Command "ShiftPosition"
  ERR_INVALID_PARAM_ROTATION_ANGLE_ONLY_MODE_3 := 16#8D67,

  /// Server Invalid parameter value - TransformationParameter_2 value does not match the selected mode
  /// Command "ShiftPosition"
  ERR_INVALID_PARAM_TRANSFORMATION_PARAM_2_INVALID := 16#8D68,

  /// Server Invalid parameter value - ToolNo outside of the allowed range 0..254 or does not exist on the RC
  /// Commands: "CalculateTool", "CalculateFrame"
  ERR_INVALID_PARAM_TOOLNO_OUT_OF_RANGE := 16#8D69,

  /// Server Invalid parameter value - FrameNo outside of the allowed range 0..254 or does not exist on the RC
  /// Command "CalculateCartesianPosition"
  ERR_INVALID_PARAM_FRAMENO_OUT_OF_RANGE := 16#8D70,

  /// Server Invalid parameter value - TargetToolNo outside of the allowed range 0..254 or does not exist on the RC
  /// Command "CalculateCartesianPosition"
  ERR_INVALID_PARAM_TARGET_TOOLNO_OUT_OF_RANGE := 16#8D71,

